// TIA Portal project "MTconnect_V15.1" (V15.1)
// demonstrates certain use cases, when migrating from Rockwell Automation to Siemens

(* hardware
DEVICE "S7-1200 station_1"  S7-1200 Station
   slot 0: "Rack_0"  S7-1200 Rack  Rack  V1.0
   slot 1: "PLC_1"  CPU 1215C AC/DC/Rly  6ES7 215-1BG40-0XB0  V4.1
*)

// ===== PLC "PLC_1"  CPU 1215C AC/DC/Rly =====
// protected blocks, not shown: "MTCONNECT", "TimeStamp"

VAR_GLOBAL   // PLC tag table "Default tag table"
   "Tag_1" AT %M5.5 : Bool;
   "RecDone" AT %M5.0 : Bool;
   "RecBusy" AT %M5.1 : Bool;
   "RecError" AT %M5.2 : Bool;
   "RecStatus" AT %MW6 : Word;
   "RecLength" AT %MW8 : Word;
   "RecTriggerSP" AT %M5.7 : Bool;
   "Clock_Byte" AT %MB0 : Byte;
   "Clock_10Hz" AT %M0.0 : Bool;
   "Clock_5Hz" AT %M0.1 : Bool;
   "Clock_2.5Hz" AT %M0.2 : Bool;
   "Clock_2Hz" AT %M0.3 : Bool;
   "Clock_1.25Hz" AT %M0.4 : Bool;
   "Clock_1Hz" AT %M0.5 : Bool;
   "Clock_0.625Hz" AT %M0.6 : Bool;
   "Clock_0.5Hz" AT %M0.7 : Bool;
   "System_Byte" AT %MB1 : Byte;
   "FirstScan" AT %M1.0 : Bool;
   "DiagStatusUpdate" AT %M1.1 : Bool;
   "AlwaysTRUE" AT %M1.2 : Bool;
   "AlwaysFALSE" AT %M1.3 : Bool;
   "Tag_2" AT %M5.6 : Bool;
   "Tag_3" AT %MD8 : UDInt;
   "Tag_4" AT %M20.0 : Bool;
   "Tag_5" AT %M20.1 : Bool;
   "Tag_6" AT %M20.2 : Bool;
   "Tag_7" AT %MW22 : Word;
   "Tag_8" AT %M20.7 : Bool;
   "Tag_9" AT %M10.7 : Bool;
   "Tag_10" AT %M10.0 : Bool;
   "Tag_11" AT %M10.1 : Bool;
   "Tag_12" AT %M10.2 : Bool;
   "Tag_13" AT %MW12 : Word;
   "SendLength" AT %MW50 : UInt;
   "Tag_15" AT %M50.1 : Bool;
   "Tag_16" AT %M52.1 : Bool;
   "Tag_17" AT %I0.0 : Bool;
   "Tag_18" AT %M15.0 : Bool;
   "SendEvent" AT %M15.1 : Bool;
   "Estop" AT %I0.2 : Bool;
   "Tag_20" AT %M15.2 : Bool;
   "Tag_21" AT %M15.3 : Bool;
   "SendPong" AT %M15.4 : Bool;
   "Tag_22" AT %M15.5 : Bool;
   "Tag_23" AT %M60.0 : Bool;
   "Tag_14" AT %M101.0 : Bool;
   "Tag_24" AT %M21.1 : Bool;
   "Tag_25" AT %MW110 : Word;
   "Tag_26" AT %M109.7 : Bool;
   "InCycle" AT %I0.3 : Bool;
   "Tag_27" AT %I0.4 : Bool;
   "Tag_28" AT %MD16 : DInt;
   "CycleCount" AT %MW20 : Int;
   "Floatnum" AT %MD24 : Real;
END_VAR

VAR_GLOBAL CONSTANT   // PLC tag table "Default tag table"
   "Constant_1" : String := 'This is constant';   // This is Comment
END_VAR

TYPE "DataItemBool"
   STRUCT
      "name" : String[20];
      category : UInt;   // 1) EVENT 2) SAMPLE 3) CONDITION
      value : Bool;
      prevValue : Bool;
      send : Bool;
   END_STRUCT;
END_TYPE

TYPE "DataItemNumeric"
   STRUCT
      "name" : String[20];
      category : UInt;   // 1) EVENT 2) SAMPLE 3) CONDITION
      value : Real;
      prevvalue : Real;
      decimal : Int;
      send : Bool;
   END_STRUCT;
END_TYPE

TYPE "DataItemString"
   STRUCT
      "name" : String[20];
      category : UInt;   // 1) EVENT 2) SAMPLE 3) CONDITION
      value : String[25];
      prevvalue : String[25];
      send : Bool;
   END_STRUCT;
END_TYPE

// folder: MTConnect

DATA_BLOCK "MTCData"   // DB4
{ S7_Optimized_Access := 'TRUE' }
VERSION : 0.1
   VAR
      "Bool" : Array[0..1] of "DataItemBool";
      Numeric : Array[0..1] of "DataItemNumeric";
      "String" : Array[0..1] of "DataItemString";
   END_VAR
BEGIN
   "Bool"[0]."name" := 'estop';
   "Bool"[0].category := 1;   // 1) EVENT 2) SAMPLE 3)CONDITION
   "Bool"[1]."name" := 'btag1';
   "Bool"[0].value := FALSE;
   "Bool"[0].prevValue := FALSE;
   "Bool"[0].send := FALSE;
   "Bool"[1].category := 0;
   "Bool"[1].value := FALSE;
   "Bool"[1].prevValue := FALSE;
   "Bool"[1].send := FALSE;
   Numeric[0]."name" := 'cycles';
   Numeric[0].category := 0;
   Numeric[0].value := 0.0;
   Numeric[0].prevvalue := 0.0;
   Numeric[0].send := FALSE;
   Numeric[1]."name" := 'ftag1';
   Numeric[1].category := 0;
   Numeric[1].value := 0.0;
   Numeric[1].prevvalue := 0.0;
   Numeric[1].send := FALSE;
END_DATA_BLOCK

// folder: (top level)

ORGANIZATION_BLOCK "Main"   // OB1, LAD, ProgramCycle
TITLE = "Main Program Sweep (Cycle)"
{ S7_Optimized_Access := 'TRUE' }
VERSION : 0.1
   VAR_INPUT
      Initial_Call : Bool;   // Initial call of this OB
      Remanence : Bool;   // =True, if remanent data are available
   END_VAR
   VAR_TEMP
      StringTemp1 : String;
      StringTemp2 : String;
   END_VAR
   VAR CONSTANT
      "TRUE/FALSE" : Bool := 1;
   END_VAR
BEGIN

REGION Network 2
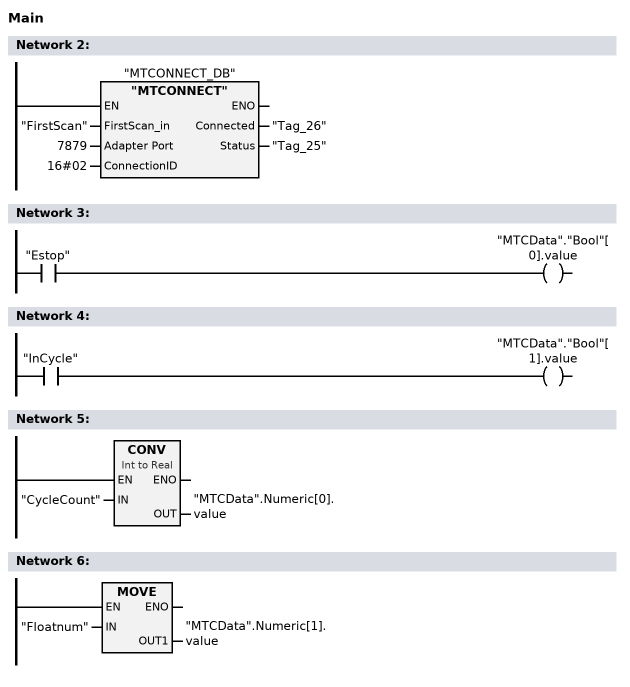
   RUNG wire#powerrail
      "MTCONNECT_DB"(FirstScan_in := "FirstScan", "Adapter Port" := 7879, ConnectionID := 16#02, Connected => "Tag_26", Status => "Tag_25")
   END_RUNG
   // the same network as SCL:
   "MTCONNECT_DB"(FirstScan_in := "FirstScan",   // "MTCONNECT"
                  "Adapter Port" := 7879,
                  ConnectionID := 16#02,
                  Connected => "Tag_26",
                  Status => "Tag_25");
END_REGION

REGION Network 3
   RUNG wire#powerrail
      Contact( "Estop" )
      Coil( "MTCData"."Bool"[0].value )
   END_RUNG
   // the same network as SCL:
   "MTCData"."Bool"[0].value := "Estop";
END_REGION

REGION Network 4
   RUNG wire#powerrail
      Contact( "InCycle" )
      Coil( "MTCData"."Bool"[1].value )
   END_RUNG
   // the same network as SCL:
   "MTCData"."Bool"[1].value := "InCycle";
END_REGION

REGION Network 5
   RUNG wire#powerrail
      { S7_Templates := "[SrcType := Int, DestType := Real]" } Convert(in := "CycleCount", out => "MTCData".Numeric[0].value)
   END_RUNG
   // the same network as SCL:
   "MTCData".Numeric[0].value := INT_TO_REAL("CycleCount");
END_REGION

REGION Network 6
   RUNG wire#powerrail
      Move(in := "Floatnum", out1 => "MTCData".Numeric[1].value)
   END_RUNG
   // the same network as SCL:
   "MTCData".Numeric[1].value := "Floatnum";
END_REGION
END_ORGANIZATION_BLOCK

ORGANIZATION_BLOCK "Data Collection"   // OB30, LAD, CyclicInterrupt
{ S7_Optimized_Access := 'TRUE' }
VERSION : 0.1
   VAR_INPUT
      Initial_Call : Bool;   // Initial call of this OB
      Event_Count : Int;   // Events discarded
   END_VAR
   VAR CONSTANT
      PI : Real := 3.14159;
   END_VAR
BEGIN

REGION Network 2
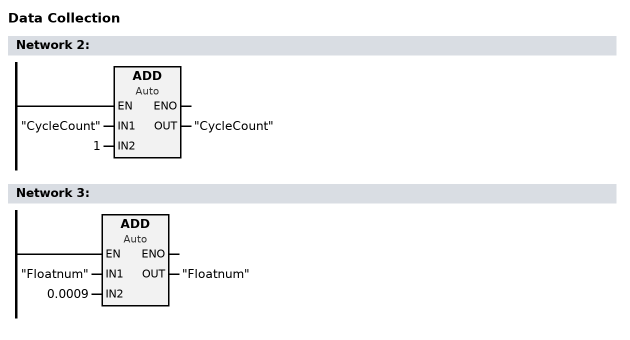
   RUNG wire#powerrail
      Add(in1 := "CycleCount", in2 := 1, out => "CycleCount")
   END_RUNG
   // the same network as SCL:
   "CycleCount" := "CycleCount" + 1;
END_REGION

REGION Network 3
   RUNG wire#powerrail
      Add(in1 := "Floatnum", in2 := 0.0009, out => "Floatnum")
   END_RUNG
   // the same network as SCL:
   "Floatnum" := "Floatnum" + 0.0009;
END_REGION
END_ORGANIZATION_BLOCK

// folder: MTConnect

FUNCTION "SizeOf" : Int   // FC4, SCL
{ S7_Optimized_Access := 'TRUE' }
VERSION : 0.1
   VAR_INPUT
      Arrayin : Variant;
   END_VAR
   VAR_TEMP
      erro : Int;
   END_VAR
BEGIN
   #SizeOf := CountOfElements(#Arrayin);
END_FUNCTION

// ===== library types =====

// folder: GET_PUT_R Datatypes

TYPE "RockwellTag"
VERSION : 0.1
   STRUCT
      ID : Int;   // [INT] TagId inside the remote PLC
      "Name" : String[24];   // [STRING24] TagName inside the remote PLC
      DataType : Int;   // [ENUM] data type of tag
      Count : Int := 1;   // [INT] number of elements to be retrieved
   END_STRUCT;
END_TYPE

TYPE "RockwellTag"
VERSION : 0.1
   STRUCT
      ID : Int;   // [INT] TagId inside the remote PLC
      "Name" : String[24];   // [STRING24] TagName inside the remote PLC
      DataType : Int;   // [ENUM] data type of tag
      Count : Int := 1;   // [INT] number of elements to be retrieved
   END_STRUCT;
END_TYPE

TYPE "RockwellConfig"
VERSION : 0.1
   STRUCT
      connID : Conn_Ouc := 0;   // [1..4096] connection identifier
      currentSessionID : UDInt;   // Session ID used for communications with Rockwell controller / currently used session ID, assigned by the remote PLC
      references : DInt;   // [0..MAX_VAR_R] number of PUT_R/ GET_R instances currently in use / reference count; 0= no connectivity
      instanceLock : DInt;   // instance number currently using send and receive capabilities
   END_STRUCT;
END_TYPE

TYPE "RockwellConfig"
VERSION : 0.1
   STRUCT
      connID : Word;   // [1..4096] connection identifier
      currentSessionID : DInt;   // Session ID used for communications with Rockwell controller / currently used session ID, assigned by the remote PLC
      references : DInt;   // [0..MAX_VAR_R] number of PUT_R/ GET_R instances currently in use / reference count; 0= no connectivity
      instanceLock : DInt;   // instance number currently using send and receive capabilities
   END_STRUCT;
END_TYPE

// folder: (top level)

FUNCTION_BLOCK "PUT_R"   // FB1, SCL
{ S7_Optimized_Access := 'FALSE' }
VERSION : 0.1
   VAR_INPUT
      Enable : Bool;   // [TRUE| FALSE] TRUE signal keeps the block in PowerOff state
      REQ : Bool;   // [TRUE |FALSE] rising edge triggers a read request
      InterfaceId : Byte;   // [1..] InterfaceID of the used interface
      IPv4 : Array[1..4] of Byte;   // [IPv4 address] - shall be in the same subnet as controller is
      Slot : Int;   // [-1..16] -1, when directly connected suc has CompactLogix
   END_VAR
   VAR_OUTPUT
      Status : Word;   // [Enum] status information
      Done : Bool;   // [TRUE | FALSE] TRUE signal is a one shot signal indicating the transmission of the data
      Connecting : Bool;   // [TRUE | FALSE] TRUE signal indicates the establishment of the connection
      Established : Bool;   // [TRUE | FALSE] TRUE indicates an established connection
   END_VAR
   VAR_IN_OUT
      Config : "RockwellConfig";
      Tag : "RockwellTag";   // [RockwelTag] datatype containing the tagname, value and data type
      Value : ANY;
   END_VAR
   VAR
      internalState : Int;   // [Enum] contains the internal state information
      connect : TCON;
      disconnect : TDISCON;
      send : TSEND;
      receive : TRCV;
      connection : TCON_PAR;
      sendBuffer : Struct
         Header : Struct
            Command : Word;   // Encapsulation command
            Length : Int;   // Length, in bytes, of the command specific data portion of the message
            SessionHandle : DInt;   // Session identification
            Status : DInt;   // Status code
            Context : Array[1..8] of Byte;   // Information pertinien only to the sender of an encapsulation command
            Options : DInt;
         END_STRUCT;
         Data : Array[1..508] of Byte;
      END_STRUCT;
      receiveBuffer : Struct
         Header : Struct
            Command : Word;   // Encapsulation command
            Length : Int;   // Length, in bytes, of the command specific data portion of the message
            SessionHandle : DInt;   // Session identification
            Status : DInt;   // Status code
            Context : Array[1..8] of Byte;   // Information pertinien only to the sender of an encapsulation command
            Options : DInt;
         END_STRUCT;
         Data : Array[1..508] of Byte;
      END_STRUCT;
      currentResponse : Word;
      connectionStatus : Struct
         isDisconnected : Bool;
         isDisconnecting : Bool;
         isConnecting : Bool;
         isConnected : Bool;
         hasReceivedData : Bool;
         hasReceivedHeader : Bool;
      END_STRUCT;
      indexTag : Int := 0;
      currentCIPService : Byte;
      previousRequest : Bool;
      EnabledJ : Bool;
      ownInstance : DInt;
      ownSequence : DInt;
      randomGenerator : Struct   // [STRUCT] used to realize a pseudo random number
         m_w : DInt;
         m_z : DInt;
         Val : DInt;
         currentTime : Date_And_Time;
         currentMilliSeconds : Time;
      END_STRUCT;
   END_VAR
   VAR_TEMP
      indexTagName : Int;
      result : Int;
      itemLength : Int;   // contains the Length of the EIP packet
      overallLength : Int;   // contains the Length of the EIP packet
      tagNameLength : Int;   // contains the Length of the Tagname (in WORDS)
      tagValueLength : Int;   // contains the Length of the Tag Value
      unconnectedDataItemLength : Int;   // contains the Length of the unconnected data item
      baseIndexOuterCIPMessage : Int;   // contains the base index to the beginning of the outer CIP message
      baseIndexInnerCIPMessage : Int;   // contains the base index to the beginning of the inner CIP message
      receivedServiceStatus : Int;
      receivedInstance : DInt;
      receivedSequence : DInt;
      receivedType : Word;
      valueIndex : Int;
      bufferIndex : Int;
      tagName : String[24];
      sendValue : Byte;
      DstAny : ANY;
      Destination AT DstAny : Struct
         ID : Byte;
         Typed : Byte;
         Amount : Int;
         Block : Int;
         Offset : Int;
      END_STRUCT;
   END_VAR
   VAR CONSTANT
      EIP_VENDOR_ID : Word := 1251;   // EtherNet/IP vendor ID 'Siemens AG'
      EIP_HEADER_LENGTH : Int := 24;   // EtherNet/IP Encapsulation Header length is 24 bytes
      EIP_PORT : Word := 44818;   // EtherNet/IP standard port is 44818 (0xAF12)
      RESULT_SUCCESS : Word := 16#0000;
      RESULT_IDLE : Word := 16#7000;
      RESULT_JOB_START : Word := 16#7001;
      RESULT_JOB_RUNNING : Word := 16#7002;
      RESULT_JOB_NOT_REQUIRED : Word := 16#80A3;
      RESULT_MORE_AVAIL : Word := 16#80B1;
      RESULT_REUSED_ID : Word := 16#8085;
      EIP_STATUS_OK : DInt := 16#0;   // EIP Status OK
      EIP_STATUS_INVALID_SESSION_ID : DInt := 16#64000000;   // EIP Status "Invalid Session ID"
      EIP_STATUS_TOOMANY_SESSIONS : DInt := 16#01000000;   // EIP Status "more than 1 active session on the same TCP connection"
      EIP_STATUS_OUTOFRESSOURCES : DInt := 16#02000000;   // EIP Status "does not have sufficient resources"
      EIP_STATUS_PROTOCOL_ERROR : DInt := 16#69000000;   // EIP Status "Protocol Version or Options mismatches"
      EIP_CMD_REG_SESSION : Word := 16#0065;   // EtherNet/IP Encapsulation Command "Register Session"
      EIP_CMD_UNREG_SESSION : Word := 16#0066;   // EtherNet/IP Encapsulation Command "Unregister Session"
      EIP_CMD_SEND_RR : Word := 16#006F;   // EtherNet/IP Encapsulation Command "Send RR Data"
      CIP_SRV_TABLEREAD : Byte := 16#4C;   // CIP Service Data Table Read
      CIP_SRV_TABLEWRITE : Byte := 16#4D;   // CIP Service Data Table Write
      CIP_SRV_TABLEREAD_FRAG : Byte := 16#52;   // CIP Service Fragmented Data Table Read
      CIP_SRV_TABLEWRITE_FRAG : Byte := 16#53;   // CIP Service Fragmented Data Table Write
      CIP_SRV_UNCONNECTED_SEND : Byte := 16#52;   // CIP Service Unconnected Send Data
      STATE_IDLE : Int := 1;
      STATE_INIT : Int := 2;
      STATE_CONNECTING : Int := 20;
      STATE_DISCONNECTING : Int := 60;
      STATE_SENDING : Int := 100;
      STATE_REGISTER_SESSION : Int := 22;
      STATE_UNREGISTER_SESSION : Int := 62;
      STATE_REGISTERING : Int := 23;
      STATE_UNREGISTERING : Int := 63;
      STATE_REGISTERED : Int := 24;
      STATE_SEND : Int := 101;
      STATE_RECEIVE_HEADER : Int := 102;
      STATE_RECEIVE_DATA : Int := 103;
      STATE_POWER_OFF : Int := 0;
      DT_BOOLEAN_ATOMIC : Int := 16#C1;
      DT_SINT_ATOMIC : Int := 16#C2;
      DT_INT_ATOMIC : Int := 16#C3;
      DT_DINT_ATOMIC : Int := 16#C4;
      DT_FLOAT_ATOMIC : Int := 16#CA;
      CIP_PATH_SEG_TYPE_CLASS : Byte := 16#20;
      CIP_PATH_SEG_TYPE_INSTANCE : Byte := 16#24;
      CIP_PATH_SEG_TYPE_ANSI : Byte := 16#91;
      CIP_PATH_SEG_TYPE_PORT : Byte := 16#01;
      CIP_ROUTE_SEG_LENGTH : Int := 4;
      CIP_ROUTE_PATH_LENGTH : Int := 1;
      CIP_TABLEREAD_LENGTH : Int := 6;
      CIP_TABLEWRITE_LENGTH : Int := 4;
      CIP_UCSEND_HEADER_LENGTH : Int := 4;
      CIP_UCSEND_SEG_LENGTH : Int := 6;
      EIP_CMD_SEND_RR_SEG_LENGTH : Int := 16;
      CON_TYPE_TCP_V2 : Byte := 16#11;
      CON_TYPE_TCP_V4 : Byte := 11;
      CIP_GENSTS_SUCCESS : Byte := 16#00;
      CIP_GENSTS_PATH_SEG_ERROR : Byte := 16#04;
      CIP_GENSTS_PATH_DEST_UNKNOWN : Byte := 16#05;
      CIP_GENSTS_PARTIAL : Byte := 16#06;
      CIP_GENSTS_NOT_ENOUGH_DATA : Byte := 16#13;
      CIP_GENSTS_PATH_SIZE_MISMATCH : Byte := 16#26;
      CIP_GENSTS_DOESNT_EXIST : Byte := 16#16;
      CIP_GENSTS_GENERIC : Byte := 16#FF;
      CIP_SRVSTS_RANGE_EXCEED : Int := 16#2105;
      CIP_SRVSTS_TYPE_MISMATCH : Int := 16#2107;
   END_VAR
BEGIN
   //=============================================================================
   // Siemens AG
   // (c)Copyright 2016 All Rights Reserved
   //-----------------------------------------------------------------------------
   // Library: PutGet_Rockwell
   // Tested with: 319F-3PN/DP V2.8.6 and ControlLogix/Compactlogix V26
   // Engineering: TIA Portal V13 SP1 Upd 9
   // Restrictions: look into pdf
   // Requirements: 
   // Functionality: Get Put Values from to Rockwell CPU
   //-----------------------------------------------------------------------------
   // Change log table:
   // Version  Date            Expert in charge        Changes applied
   // 01.00.00 12.07.2016      Scheel                  initial version 
   // 01.00.01 20.10.2016      Scheel                  feat: add diagnostics and
   //                                                        indicators
   //                                                  style: remove duplicate
   //                                                         code segments
   //                                                  fix: connect will be
   //                                                       retriggered, when idle
   //                                                  refac: change of IP address
   //                                                         datatype to IP_V4
   //                                                  feat: add recognition of
   //                                                        CIP specific status
   //
   //#########################################################################################
   // Pseudo Random number generator
   //
   //  This Random number function generator is based on multiplication and
   //  addition with overflow invented by George Marsaglia.
   //  The loss of information is intended.
   //  
   //  Wikipedia (https://en.wikipedia.org/wiki/Random_number_generation)
   //#########################################################################################
   //
   //Initialization of the variables using a time value as a seed
   #randomGenerator.currentMilliSeconds := TIME_TCK();

   IF #randomGenerator.m_w = 0 OR #randomGenerator.m_z = 0 THEN
     #randomGenerator.m_w := T_CONV(TIME_TCK());    // using the milliseconds since the PLC has been powered on
     #randomGenerator.m_z := 13696;
   ELSE
     #randomGenerator.m_z := 36969 * DWORD_TO_DINT(DINT_TO_DWORD(#randomGenerator.m_z) AND 16#FFFF)
     + DWORD_TO_DINT(SHR(IN := DINT_TO_DWORD(#randomGenerator.m_z), N := 16));
     #randomGenerator.m_w := 18000 * DWORD_TO_DINT(DINT_TO_DWORD(#randomGenerator.m_w) AND 16#FFFF)
     + DWORD_TO_DINT(SHR(IN := DINT_TO_DWORD(#randomGenerator.m_w), N := 16));
     #randomGenerator.Val := DWORD_TO_DINT(SHL(IN := DINT_TO_DWORD(#randomGenerator.m_z), N := 16)) + #randomGenerator.m_w;  // 32-bit result */    
   END_IF;

   //assume sane state
   #Status := #RESULT_IDLE;
   #Done := FALSE;

   #connect(ID := #connection.id,
            CONNECT := #connection);

   #disconnect(ID := #connection.id);


   IF NOT #Enable AND #EnabledJ THEN
     // Complete Restart detected 
     //
     #internalState := #STATE_UNREGISTER_SESSION;

   ELSIF #Enable AND NOT #EnabledJ THEN
     #internalState := #STATE_INIT;

   ELSE
     // Regular operation
     //   
     CASE #internalState OF
       #STATE_POWER_OFF:
         //Preset the TCP connection information
         //  
         IF #Config.connID = 0 THEN
           #Config.connID := DWORD_TO_WORD(DINT_TO_DWORD((#randomGenerator.Val MOD 2048) + 2048));
         END_IF;
         #connection.id := #Config.connID;

         #connection.connection_type := #CON_TYPE_TCP_V2;      //TCP connection
         #connection.local_device_id := #InterfaceId;
         #connection.active_est := TRUE;                //active connection (Client)

         #connection.local_tsap_id_len := 0;

         #connection.rem_staddr_len := 4;
         #connection.rem_staddr[1] := #IPv4[1];
         #connection.rem_staddr[2] := #IPv4[2];
         #connection.rem_staddr[3] := #IPv4[3];
         #connection.rem_staddr[4] := #IPv4[4];

         #connection.rem_tsap_id_len := 2;
         #connection.rem_tsap_id[1] := WORD_TO_BYTE(SHR(IN := #EIP_PORT, N := 8));
         #connection.rem_tsap_id[2] := WORD_TO_BYTE(#EIP_PORT AND W#16#FF);

         #ownInstance := 0;
         #ownSequence := 0;

         #internalState := #STATE_IDLE;

       #STATE_IDLE:

         // Action
         // 
         #Done := FALSE;

         // Transition 
         //IF NOT #connectionStatus.isConnected THEN
         //  #internalState := #STATE_INIT;          
         IF #connectionStatus.isConnected AND #REQ AND NOT #previousRequest AND #Enable THEN
           #internalState := #STATE_SENDING;
           #Status := #RESULT_JOB_START;
         END_IF;


       #STATE_INIT:
         //Preset the TCP connection information
         //
         IF #Config.connID = 0 THEN
           #Config.connID := DWORD_TO_WORD(DINT_TO_DWORD((#randomGenerator.Val MOD 2048) + 2048));
         END_IF;
         #connection.id := #Config.connID;

         //Inserting Semaphore checking
         //
         //  Only issue a new connect, when there is no one is referencing the connection already
         //  Otherwise just skip that step and use the established connection
         //  

         IF #Config.references = 0 THEN
           #connection.connection_type := #CON_TYPE_TCP_V2;      //TCP connection
           #connection.local_device_id := #InterfaceId;
           #connection.active_est := TRUE;                //active connection (Client)

           #connection.local_tsap_id_len := 0;

           #connection.rem_staddr_len := 4;
           #connection.rem_staddr[1] := #IPv4[1];
           #connection.rem_staddr[2] := #IPv4[2];
           #connection.rem_staddr[3] := #IPv4[3];
           #connection.rem_staddr[4] := #IPv4[4];

           #connection.rem_tsap_id_len := 2;
           #connection.rem_tsap_id[1] := WORD_TO_BYTE(SHR(IN := #EIP_PORT, N := 8));
           #connection.rem_tsap_id[2] := WORD_TO_BYTE(#EIP_PORT AND W#16#FF);


           //No connection established yet
           //  issue a new request
           #connect.REQ := TRUE;
           #internalState := #STATE_CONNECTING;
         ELSE
           #internalState := #STATE_IDLE;
           #connectionStatus.isConnected := TRUE;
         END_IF;
         #Config.references := #Config.references + 1;

         //Remember the currently active instance reference as my own instance identifier
         //  and reset the Sequence counter
         #ownInstance := #Config.references;
         #ownSequence := 0;

       #STATE_CONNECTING:

         IF #connect.STATUS = #RESULT_JOB_START THEN
           #connectionStatus.isConnecting := TRUE;

         ELSIF #connect.STATUS = #RESULT_IDLE THEN
           #connect.REQ := NOT #connect.REQ;

         ELSIF #connect.STATUS = #RESULT_JOB_RUNNING THEN
           #connect.REQ := FALSE;

         ELSIF #connect.STATUS = #RESULT_JOB_NOT_REQUIRED OR
           #connect.STATUS = #RESULT_SUCCESS
         THEN
           #connect.REQ := FALSE;
           #connectionStatus.isConnecting := FALSE;
           #connectionStatus.isConnected := TRUE;
           #connectionStatus.isDisconnected := FALSE;

           #internalState := #STATE_REGISTER_SESSION;

         ELSE
           // Throw error !
           //   Error in connect
           #Status := W#16#8100 OR (#connect.STATUS AND 16#00FF);   //Error in connecting       
           #connect.REQ := FALSE;
           #internalState := #STATE_DISCONNECTING;
         END_IF;

       #STATE_REGISTER_SESSION:

         // SWAP (W#16#AFCD) = W#16#CDAF
         // 
         //  SHL(AFCD, 8) OR SHR(AFCD, 8)

         #sendBuffer.Header.Command := (SHL(IN := #EIP_CMD_REG_SESSION, N := 8) OR SHR(IN := #EIP_CMD_REG_SESSION, N := 8)); //Command is RegisterSession (16#65)
         #sendBuffer.Header.Length := WORD_TO_INT(W#16#0400);          //Length of Data is 4 Bytes
         #sendBuffer.Header.SessionHandle := 0;
         #sendBuffer.Header.Status := 0;
         #sendBuffer.Header.Options := 0;
         //the Context will be a combination out of the own instance identifier
         //and a sequence number
         #sendBuffer.Header.Context[1] := DWORD_TO_BYTE(DINT_TO_DWORD(#ownInstance) AND DW#16#000000FF);
         #sendBuffer.Header.Context[2] := DWORD_TO_BYTE(SHR(IN := DINT_TO_DWORD(#ownInstance), N := 8) AND DW#16#000000FF);
         #sendBuffer.Header.Context[3] := DWORD_TO_BYTE(SHR(IN := DINT_TO_DWORD(#ownInstance), N := 16) AND DW#16#000000FF);
         #sendBuffer.Header.Context[4] := DWORD_TO_BYTE(SHR(IN := DINT_TO_DWORD(#ownInstance), N := 24) AND DW#16#000000FF);
         #sendBuffer.Header.Context[5] := DWORD_TO_BYTE(DINT_TO_DWORD(#ownSequence) AND DW#16#000000FF);
         #sendBuffer.Header.Context[6] := DWORD_TO_BYTE(SHR(IN := DINT_TO_DWORD(#ownSequence), N := 8) AND DW#16#000000FF);
         #sendBuffer.Header.Context[7] := DWORD_TO_BYTE(SHR(IN := DINT_TO_DWORD(#ownSequence), N := 16) AND DW#16#000000FF);
         #sendBuffer.Header.Context[8] := DWORD_TO_BYTE(SHR(IN := DINT_TO_DWORD(#ownSequence), N := 24) AND DW#16#000000FF);
         #sendBuffer.Data[1] := 16#01;                                 //Protocol Version V1.0

         //Checking the MuteEx
         IF #Config.instanceLock = 0 OR
           #Config.instanceLock = #ownInstance
         THEN
           //allowed to utilize, since instanceLock is either 0 or ownInstance
           #send(ID := #connection.id,
                 DATA := #sendBuffer);

           //Locking the MutEx
           #Config.instanceLock := #ownInstance;
           #send.LEN := #EIP_HEADER_LENGTH + 4;
           #send.REQ := TRUE;

           #internalState := #STATE_REGISTERING;
         ELSE
           ;
         END_IF;

       #STATE_REGISTERING:
         // Action
         // 

         //allowed to utilize, since instanceLock is either 0 or ownInstance
         #send(ID := #connection.id,
               DATA := #sendBuffer);

         // Transition
         // 
         IF #send.STATUS = #RESULT_JOB_START THEN
           ;
         ELSIF #send.STATUS = #RESULT_JOB_RUNNING THEN
           #send.REQ := FALSE;

         ELSIF #send.STATUS = #RESULT_IDLE THEN
           #send.REQ := NOT #send.REQ;

         ELSIF #send.STATUS = #RESULT_SUCCESS THEN
           #send.REQ := FALSE;
           #internalState := #STATE_RECEIVE_HEADER;
         ELSE
           // Throw error !
           //   in Registering
           #Status := W#16#8200 OR (#send.STATUS AND 16#00FF);   //Error in sending
           #send.REQ := FALSE;
           #internalState := #STATE_DISCONNECTING;
         END_IF;

       #STATE_SENDING:
         #sendBuffer.Header.Command := (SHL(IN := #EIP_CMD_SEND_RR, N := 8) OR SHR(IN := #EIP_CMD_SEND_RR, N := 8));       //Command is SendRRData (16#6F)
         //
         // overall Message length depends on the packet content and is therefore assigned later
         //
         // SWAP (DW#16#0102ABCD) = CDAB0201
         // 
         //   = SHL(<value>,24) OR (SHL(<value>, 8) AND DW#16#00FF0000) OR (SHR(<value>, 8) AND DW#16#0000FF00) OR SHR(<value>,24)

         //#sendBuffer.Header.SessionHandle := DWORD_TO_DINT(SWAP(DINT_TO_DWORD(#Config.currentSessionID)));
         #sendBuffer.Header.SessionHandle := DWORD_TO_DINT(SHL(IN := DINT_TO_DWORD(#Config.currentSessionID), N := 24) OR
                                                           (SHL(IN := DINT_TO_DWORD(#Config.currentSessionID), N := 8) AND DW#16#00FF0000) OR
                                                           (SHR(IN := DINT_TO_DWORD(#Config.currentSessionID), N := 8) AND DW#16#0000FF00) OR
                                                           SHR(IN := DINT_TO_DWORD(#Config.currentSessionID), N := 24));

         ;
         #sendBuffer.Header.Status := 0;
         #sendBuffer.Header.Options := 0;
         //the Context will be a combination out of the own instance identifier
         //and a sequence number
         #sendBuffer.Header.Context[1] := DWORD_TO_BYTE(DINT_TO_DWORD(#ownInstance) AND DW#16#000000FF);
         #sendBuffer.Header.Context[2] := DWORD_TO_BYTE(SHR(IN := DINT_TO_DWORD(#ownInstance), N := 8) AND DW#16#000000FF);
         #sendBuffer.Header.Context[3] := DWORD_TO_BYTE(SHR(IN := DINT_TO_DWORD(#ownInstance), N := 16) AND DW#16#000000FF);
         #sendBuffer.Header.Context[4] := DWORD_TO_BYTE(SHR(IN := DINT_TO_DWORD(#ownInstance), N := 24) AND DW#16#000000FF);
         #sendBuffer.Header.Context[5] := DWORD_TO_BYTE(DINT_TO_DWORD(#ownSequence) AND DW#16#000000FF);
         #sendBuffer.Header.Context[6] := DWORD_TO_BYTE(SHR(IN := DINT_TO_DWORD(#ownSequence), N := 8) AND DW#16#000000FF);
         #sendBuffer.Header.Context[7] := DWORD_TO_BYTE(SHR(IN := DINT_TO_DWORD(#ownSequence), N := 16) AND DW#16#000000FF);
         #sendBuffer.Header.Context[8] := DWORD_TO_BYTE(SHR(IN := DINT_TO_DWORD(#ownSequence), N := 24) AND DW#16#000000FF);
         //CIP specific data
         #sendBuffer.Data[1] := 16#0;                                 //CIP Interface handle
         #sendBuffer.Data[2] := 16#0;
         #sendBuffer.Data[3] := 16#0;
         #sendBuffer.Data[4] := 16#0;

         #sendBuffer.Data[5] := 16#0;                                  //Timeout
         #sendBuffer.Data[6] := 16#0;

         #sendBuffer.Data[7] := 16#2;                                  //Items
         #sendBuffer.Data[8] := 16#0;

         #sendBuffer.Data[9] := 16#0;                                  //Null address item
         #sendBuffer.Data[10] := 16#0;
         #sendBuffer.Data[11] := 16#0;                                  //Null address item Length = 0
         #sendBuffer.Data[12] := 16#0;

         #sendBuffer.Data[13] := 16#B2;                                  //Unconnected data item
         #sendBuffer.Data[14] := 16#0;
         //Item Length needs to be added, but since that depends on the content,
         //it will will be assigned later. It occupies 2 Bytes, thus the outer CIP Message 
         //starts at offset 17 into the Data (1 based counting)
         //
         #baseIndexOuterCIPMessage := 17;

         //CIP Message
         //  here a decision needs to be made
         //  In case Slot is -1 a direct connection is assumed, such as for a CompactLogix, this means no
         //  further route segments are necessary
         //  In case Slot is anywhere between 0 and 16 a route segment is required, since the CPU is not
         //  identical to the ethernet interface, as in a ControlLogix L5, L6, L7 series system

         //Length of the following Path segment depends only on the length of the Tagname measured in WORDS
         // plus 1 WORD for the segment encoding information
         // 
         #tagName := #Tag."Name";
         #tagNameLength := ((LEN(#tagName) + 1) / 2) * 2;

         //
         //  Prelude
         //
         //In case the slot information is negative (-1) there is no additional path segment
         //Any other slot value requires routing information, which need to be added
         //  this means the preparation of offsets and header needs to be done, before
         //  the common part of copying the value to the packet can take place
         IF #Slot = -1 THEN
           //directly connected (onboard) Ethernet interface
           //
           #baseIndexInnerCIPMessage := #baseIndexOuterCIPMessage;

         ELSE
           //not directly connected (through external) Ethernet interface
           //
           //  preparing offsets for length calculation as well as header
           //  There is a 10 byte segment before the tag value segment
           #baseIndexInnerCIPMessage := #baseIndexOuterCIPMessage + 10;

           #sendBuffer.Data[#baseIndexOuterCIPMessage] := #CIP_SRV_UNCONNECTED_SEND;                //CIP service = UNCONNECTED_SEND_DATA = 16#52
           #sendBuffer.Data[#baseIndexOuterCIPMessage + 1] := 2;                                    //Path Size is constant 2 WORDS

           #sendBuffer.Data[#baseIndexOuterCIPMessage + 2] := #CIP_PATH_SEG_TYPE_CLASS;             //Path Type = Class Segment
           #sendBuffer.Data[#baseIndexOuterCIPMessage + 3] := 16#06;                                //Class = ConnectionManager (16#06)

           #sendBuffer.Data[#baseIndexOuterCIPMessage + 4] := #CIP_PATH_SEG_TYPE_INSTANCE;          //Path Type = Instance Segment
           #sendBuffer.Data[#baseIndexOuterCIPMessage + 5] := 16#01;                                //Instance =Instance 1 (16#01)

           //Encapsulated CIP Message
           //
           #sendBuffer.Data[#baseIndexOuterCIPMessage + 6] := 16#07;                                //Priority combined with TimeTick (= 16#07)
           #sendBuffer.Data[#baseIndexOuterCIPMessage + 7] := INT_TO_BYTE(233);                     //???

         END_IF;

         //
         // tag value segment
         // 

         #sendBuffer.Data[#baseIndexInnerCIPMessage] := #CIP_SRV_TABLEWRITE;                        //CIP service = DATA_TABLE_READ = 16#4D

         #sendBuffer.Data[#baseIndexInnerCIPMessage + 1] := DINT_TO_BYTE(#tagNameLength / 2 + 1);  //Path Size
         #sendBuffer.Data[#baseIndexInnerCIPMessage + 2] := #CIP_PATH_SEG_TYPE_ANSI;                //Path Type = ANSI Extended Symbol Segment

         //Copy In
         //
         #tagName := #Tag."Name";
         #sendBuffer.Data[#baseIndexInnerCIPMessage + 3] := INT_TO_BYTE(LEN(#tagName));   //TagName Length (bytes)
         FOR #indexTagName := 1 TO BYTE_TO_INT(#sendBuffer.Data[#baseIndexInnerCIPMessage + 3]) DO
           #sendBuffer.Data[#baseIndexInnerCIPMessage + 3 + #indexTagName] := CHAR_TO_BYTE(S_CONV(MID(IN := #tagName, L := 1, P := #indexTagName)));
         END_FOR;
         //in case the tag name has an odd (uneven) length the path segment content needs to be padded to be WORD aligned
         //
         #indexTagName := #indexTagName - 1;
         IF #indexTagName MOD 2 <> 0 THEN
           #indexTagName := #indexTagName + 1;
           #sendBuffer.Data[#baseIndexInnerCIPMessage + 3 + #indexTagName] := 0;
         END_IF;

         //Command Specific information
         //
         #sendBuffer.Data[#baseIndexInnerCIPMessage + 4 + #indexTagName] := INT_TO_BYTE(#Tag.DataType);
         #sendBuffer.Data[#baseIndexInnerCIPMessage + 5 + #indexTagName] := 0;
         #sendBuffer.Data[#baseIndexInnerCIPMessage + 6 + #indexTagName] := INT_TO_BYTE(#Tag.Count);                 //number of values to follow
         #sendBuffer.Data[#baseIndexInnerCIPMessage + 7 + #indexTagName] := WORD_TO_BYTE(SHR(IN := INT_TO_WORD(#Tag.Count), N := 8) AND W#16#00FF);

         #bufferIndex := #baseIndexInnerCIPMessage + 8 + #indexTagName;

         #DstAny := #sendBuffer.Data[#bufferIndex];
         #Destination.Amount := #Tag.Count;

         //Copy the value in, type dependant
         CASE #Tag.DataType OF
           #DT_BOOLEAN_ATOMIC:
             //Transferring the Value
             //
             // Adjust the type
             #Destination.Typed := B#16#02;


             #result := BLKMOV(SRCBLK := #Value,
                               DSTBLK => #DstAny);

             #tagValueLength := 4 + #Tag.Count * 1;
           #DT_SINT_ATOMIC:
             //Transferring the Value
             //
             // Adjust the type
             #Destination.Typed := B#16#02;

             #result := BLKMOV(SRCBLK := #Value,
                               DSTBLK => #DstAny);
             #tagValueLength := 4 + #Tag.Count * 1;
           #DT_INT_ATOMIC:
             //Transferring the Value
             //
             // Adjust the type
             #Destination.Typed := B#16#05;

             #result := BLKMOV(SRCBLK := #Value,
                               DSTBLK => #DstAny);

             // Swapping the bytes for each value
             // 
             #valueIndex := 0;

             WHILE #valueIndex <= #Tag.Count DO
               #sendValue                                           := #sendBuffer.Data[#bufferIndex + 1 + 2 * #valueIndex];
               #sendBuffer.Data[#bufferIndex + 1 + 2 * #valueIndex] := #sendBuffer.Data[#bufferIndex     + 2 * #valueIndex];
               #sendBuffer.Data[#bufferIndex     + 2 * #valueIndex] := #sendValue;
               #valueIndex := #valueIndex + 1;
             END_WHILE;

             #tagValueLength := 4 + #Tag.Count * 2;
           #DT_DINT_ATOMIC:
             //Transferring the Value
             //
             // Adjust the type
             #Destination.Typed := B#16#07;

             #result := BLKMOV(SRCBLK := #Value,
                               DSTBLK => #DstAny);

             #valueIndex := 0;
             WHILE #valueIndex <= #Tag.Count DO

               // swap the received value
               #sendValue                                           := #sendBuffer.Data[#bufferIndex + 3 + 2 * #valueIndex];
               #sendBuffer.Data[#bufferIndex + 3 + 2 * #valueIndex] := #sendBuffer.Data[#bufferIndex     + 2 * #valueIndex];
               #sendBuffer.Data[#bufferIndex     + 2 * #valueIndex] := #sendValue;

               #sendValue                                           := #sendBuffer.Data[#bufferIndex + 2 + 2 * #valueIndex];
               #sendBuffer.Data[#bufferIndex + 2 + 2 * #valueIndex] := #sendBuffer.Data[#bufferIndex + 1 + 2 * #valueIndex];
               #sendBuffer.Data[#bufferIndex + 1 + 2 * #valueIndex] := #sendValue;

               #valueIndex := #valueIndex + 1;
             END_WHILE;

             #tagValueLength := 4 + #Tag.Count * 4;
           #DT_FLOAT_ATOMIC:
             //Transferring the Value
             //
             // Adjust the type
             #Destination.Typed := B#16#08;

             #result := BLKMOV(SRCBLK := #Value,
                               DSTBLK => #DstAny);

             #valueIndex := 0;
             WHILE #valueIndex <= #Tag.Count DO

               // swap the received value
               #sendValue                                           := #sendBuffer.Data[#bufferIndex + 3 + 2 * #valueIndex];
               #sendBuffer.Data[#bufferIndex + 3 + 2 * #valueIndex] := #sendBuffer.Data[#bufferIndex     + 2 * #valueIndex];
               #sendBuffer.Data[#bufferIndex     + 2 * #valueIndex] := #sendValue;

               #sendValue                                           := #sendBuffer.Data[#bufferIndex + 2 + 2 * #valueIndex];
               #sendBuffer.Data[#bufferIndex + 2 + 2 * #valueIndex] := #sendBuffer.Data[#bufferIndex + 1 + 2 * #valueIndex];
               #sendBuffer.Data[#bufferIndex + 1 + 2 * #valueIndex] := #sendValue;

               #valueIndex := #valueIndex + 1;
             END_WHILE;

             #tagValueLength := 4 + #Tag.Count * 4;
         ELSE

           //Throw error
           //  - unknown/ unsupported data type specified
           //  
           // throw warning
           #Status := 16#71A3; //Unknown data type
           #tagValueLength := 0;
         END_CASE;

         #itemLength := #tagNameLength + #tagValueLength + #CIP_TABLEWRITE_LENGTH;

         //
         // Closure
         //

         IF #Slot = -1 THEN
           #unconnectedDataItemLength := #itemLength;
         ELSE
           #sendBuffer.Data[#baseIndexOuterCIPMessage + 8] := WORD_TO_BYTE(DINT_TO_WORD(#itemLength));                  //Unconnected data item Length
           #sendBuffer.Data[#baseIndexOuterCIPMessage + 9] := WORD_TO_BYTE(SHL(IN := DINT_TO_WORD(#itemLength), N := 8));  //Unconnected data item Length

           //Routing Information
           #sendBuffer.Data[#baseIndexInnerCIPMessage + #itemLength] := INT_TO_BYTE(#CIP_ROUTE_PATH_LENGTH);
           #sendBuffer.Data[#baseIndexInnerCIPMessage + #itemLength + 1] := 0;

           #sendBuffer.Data[#baseIndexInnerCIPMessage + #itemLength + 2] := #CIP_PATH_SEG_TYPE_PORT;
           #sendBuffer.Data[#baseIndexInnerCIPMessage + #itemLength + 3] := INT_TO_BYTE(#Slot);



           #unconnectedDataItemLength :=   #itemLength
                                         + #CIP_ROUTE_SEG_LENGTH
                                         + #CIP_UCSEND_HEADER_LENGTH
                                         + #CIP_UCSEND_SEG_LENGTH;
         END_IF;

         //Length of the unconnected data item depends on the content of the package
         //
         #sendBuffer.Data[15] := WORD_TO_BYTE(DINT_TO_WORD(#unconnectedDataItemLength));        //Unconnected data item Length
         #sendBuffer.Data[16] := WORD_TO_BYTE(SHL(IN := DINT_TO_WORD(#unconnectedDataItemLength), N := 8));  //Unconnected data item Length


         #sendBuffer.Header.Length := WORD_TO_INT(SHL(IN := INT_TO_WORD(#unconnectedDataItemLength + #EIP_CMD_SEND_RR_SEG_LENGTH), N := 8) OR
                                                  SHR(IN := INT_TO_WORD(#unconnectedDataItemLength + #EIP_CMD_SEND_RR_SEG_LENGTH), N := 8));    //Length of Data

         //Checking the MuteEx
         IF #Config.instanceLock = 0 OR
           #Config.instanceLock = #ownInstance
         THEN
           #Config.instanceLock := #ownInstance;
           #send.LEN := DINT_TO_INT(#EIP_HEADER_LENGTH + #unconnectedDataItemLength + #EIP_CMD_SEND_RR_SEG_LENGTH);
           #send.REQ := TRUE;

           #ownSequence := #ownSequence + 1;
           //allowed to utilize, since instanceLock is either 0 or ownInstance
           #send(ID := #connection.id,
                 DATA := #sendBuffer);

           #internalState := #STATE_SEND;
         ELSE
           ;
         END_IF;
         #Status := #RESULT_JOB_RUNNING;

       #STATE_SEND:
         // Action
         // 

         // assume job is still running
         #Status := #RESULT_JOB_RUNNING;

         #send(ID := #connection.id,
               DATA := #sendBuffer);

         // Transition
         //
         IF #send.STATUS = #RESULT_JOB_START THEN
           ;
         ELSIF #send.STATUS = #RESULT_IDLE THEN
           #send.REQ := NOT #send.REQ;

         ELSIF #send.STATUS = #RESULT_JOB_RUNNING THEN
           #send.REQ := FALSE;

         ELSIF #send.STATUS = #RESULT_SUCCESS THEN
           #send.REQ := FALSE;
           #internalState := #STATE_RECEIVE_HEADER;
         ELSE
           // Throw error !
           // 
            #Status := W#16#8200 OR (#send.STATUS AND 16#00FF);
           #send.REQ := FALSE;
           #internalState := #STATE_DISCONNECTING;
         END_IF;

       #STATE_RECEIVE_HEADER:
         // Action
         // Receive Header data
         // 

         // assume job is still running
         #Status := #RESULT_JOB_RUNNING;

         #receive(EN_R := (#ownInstance = #Config.instanceLock),
                  ID := #connection.id,
                  LEN := #EIP_HEADER_LENGTH,
                  DATA := #receiveBuffer.Header);


         // Transition
         // Header received --> STATE_RECEIVE_DATA
         // Invalid Data --> IDLE
         // Error --> INIT
         IF #receive.NDR OR #receive.STATUS = #RESULT_SUCCESS THEN
           IF #receiveBuffer.Header.Length = 0 THEN
             //Unlocking MuteEx
             #Config.instanceLock := 0;
             #internalState := #STATE_IDLE;
           ELSE
             #internalState := #STATE_RECEIVE_DATA;
           END_IF;
         ELSIF #receive.STATUS <> #RESULT_IDLE AND
           #receive.STATUS <> #RESULT_JOB_RUNNING AND
           #receive.STATUS <> #RESULT_JOB_START AND
           #receive.STATUS <> #RESULT_SUCCESS
         THEN
           #Status := W#16#8300 OR (#receive.STATUS AND 16#00FF);
           #internalState := #STATE_IDLE;
         ELSE
           //Nothing to do, just wait here
           ;
         END_IF;

       #STATE_RECEIVE_DATA:
         // Action
         // Receive Data
         // 
         // assume job is still running
         #Status := #RESULT_JOB_RUNNING;

         #receive(EN_R := (#ownInstance = #Config.instanceLock),
                  ID := #connection.id,
                  LEN := WORD_TO_INT((SHL(IN:=INT_TO_WORD(#receiveBuffer.Header.Length),N:= 8) OR
                                      SHR(IN:=INT_TO_WORD(#receiveBuffer.Header.Length),N:= 8))),
                  DATA := #receiveBuffer.Data);

         // Transition
         // Header received --> STATE_RECEIVE_DATA
         // Invalid Data --> IDLE
         // Error --> INIT
         IF #receive.NDR OR #receive.STATUS = #RESULT_SUCCESS THEN
           // Decode Response
           // 
           #currentResponse := (SHL(IN:=#receiveBuffer.Header.Command, N:=8) OR
                                SHR(IN:=#receiveBuffer.Header.Command, N:=8));

           //the Context will be a combination out of the own instance identifier
           //and a sequence number
           #receivedInstance := DWORD_TO_DINT(SHL(IN := BYTE_TO_DWORD(#receiveBuffer.Header.Context[4]), N := 24) OR
                                              SHL(IN := BYTE_TO_DWORD(#receiveBuffer.Header.Context[3]), N := 16) OR
                                              SHL(IN := BYTE_TO_DWORD(#receiveBuffer.Header.Context[2]), N := 8) OR
                                              BYTE_TO_DWORD(#receiveBuffer.Header.Context[1]));

           #receivedSequence := DWORD_TO_DINT(SHL(IN := BYTE_TO_DWORD(#receiveBuffer.Header.Context[8]), N := 24) OR
                                              SHL(IN := BYTE_TO_DWORD(#receiveBuffer.Header.Context[7]), N := 16) OR
                                              SHL(IN := BYTE_TO_DWORD(#receiveBuffer.Header.Context[6]), N := 8) OR
                                              BYTE_TO_DWORD(#receiveBuffer.Header.Context[5]));

           IF #currentResponse = #EIP_CMD_REG_SESSION THEN
             //Response to RegisterSession received
             // retrieve the SessionID (SessionHandle)
             IF #receiveBuffer.Header.Status = #EIP_STATUS_OK THEN
               #Config.currentSessionID := DWORD_TO_DINT(SHL(IN := DINT_TO_DWORD(#receiveBuffer.Header.SessionHandle), N := 24) OR
                                                         (SHL(IN := DINT_TO_DWORD(#receiveBuffer.Header.SessionHandle), N := 8) AND DW#16#00FF0000) OR
                                                         (SHR(IN := DINT_TO_DWORD(#receiveBuffer.Header.SessionHandle), N := 8) AND DW#16#0000FF00) OR
                                                         SHR(IN := DINT_TO_DWORD(#receiveBuffer.Header.SessionHandle), N := 24));
               #Status := #RESULT_SUCCESS;
             ELSE
               // inform the user about it
               //
               #Status := W#16#7100 OR DWORD_TO_WORD((SHR(IN := DINT_TO_DWORD(#receiveBuffer.Header.Status), N := 24)));

               //Cleaning up internal information and
               //gracefully disconnect
               IF #Config.currentSessionID = 0 THEN
                 // a previous session hasn't been established --> only disconnecting
                 #internalState := #STATE_DISCONNECTING;
               ELSE
                 // previous session existed (somehow) --> unregister before disconnecting
                 #internalState := #STATE_UNREGISTER_SESSION;
               END_IF;
             END_IF;

           ELSIF #currentResponse = #EIP_CMD_SEND_RR THEN
             //Response to Send RR Data received
             // determine Status of transmission
             // retrieve TagValue and DataType
             IF #receiveBuffer.Header.Status = #EIP_STATUS_OK THEN
               #itemLength := WORD_TO_INT(SHL(IN := BYTE_TO_WORD(#receiveBuffer.Data[16]), N := 8) OR BYTE_TO_WORD(#receiveBuffer.Data[15]));
               #currentCIPService := #receiveBuffer.Data[17];
               IF #currentCIPService = (#CIP_SRV_TABLEWRITE OR 16#80) AND
                 #receivedInstance = #ownInstance AND
                 #receivedSequence = #ownSequence
               THEN
                 #ownSequence := #ownSequence + 1;

                 IF #receiveBuffer.Data[19] = #CIP_GENSTS_SUCCESS THEN
                   #Status := #RESULT_SUCCESS;
                   #Done := TRUE;

                 ELSIF #receiveBuffer.Data[19] = #CIP_GENSTS_PATH_DEST_UNKNOWN OR
                       #receiveBuffer.Data[19] = #CIP_GENSTS_PATH_SEG_ERROR
                 THEN
                   // throw warning
                   #Status := W#16#7200 OR #receiveBuffer.Data[19];

                 ELSIF #receiveBuffer.Data[19] = #CIP_GENSTS_GENERIC THEN
                   #Status := W#16#7300 OR #receiveBuffer.Data[21];
                 ELSE
                   // throw warning
                   #Status := W#16#72FF;  //Unknown error code
                 END_IF;

               ELSIF #currentCIPService = (#CIP_SRV_TABLEWRITE_FRAG OR 16#80) THEN
                 #Status := W#16#7300 OR #receiveBuffer.Data[19];

               ELSE
                 // throw warning
                 //   unexpected answer from host - ignoring it
                 #Status := W#16#8A00 OR #currentCIPService;
               END_IF;

             ELSE
               // inform the user about it
               //
               #Status := W#16#7100 OR DWORD_TO_WORD((SHR(IN := DINT_TO_DWORD(#receiveBuffer.Header.Status), N := 24)));

               //Cleaning up internal information and
               //gracefully disconnect
               IF #Config.currentSessionID = 0 THEN
                   // a previous session hasn't been established --> only disconnecting
                   #internalState := #STATE_DISCONNECTING;
                 ELSE
                   // previous session existed (somehow) --> unregister before disconnecting
                   #internalState := #STATE_UNREGISTER_SESSION;
                 END_IF;
             END_IF;
           ELSE
             //Unknown/ Unhandled Response received
             //  ignoring it
             #Status := W#16#8B00 OR #currentResponse;
             //#Config.currentSessionID := 0;
             //#internalState := #STATE_DISCONNECTING;
           END_IF;

           #receiveBuffer.Header.Length := 0;

           //Unlocking MuteEx
           #Config.instanceLock := 0;

           #internalState := #STATE_IDLE;

         ELSIF #receive.STATUS <> #RESULT_IDLE AND
           #receive.STATUS <> #RESULT_JOB_RUNNING AND
           #receive.STATUS <> #RESULT_JOB_START AND
           #receive.STATUS <> #RESULT_SUCCESS
         THEN
           #Status := W#16#8300 OR (#receive.STATUS AND 16#00FF);
           #internalState := #STATE_IDLE;
         ELSE
           ;
         END_IF;

       #STATE_UNREGISTER_SESSION:
         IF #Config.references = 1 THEN

           #sendBuffer.Header.Command := SHL(IN := #EIP_CMD_UNREG_SESSION, N := 8) OR
           SHR(IN := #EIP_CMD_UNREG_SESSION, N := 8);   //Command is RegisterSession (16#66)
           #sendBuffer.Header.Length := WORD_TO_INT(SHL(IN := INT_TO_WORD(#send.LEN - #EIP_HEADER_LENGTH), N := 8) OR
                                                    SHR(IN := INT_TO_WORD(#send.LEN - #EIP_HEADER_LENGTH), N := 8));    //Length of Data is 4 Bytes

           // SWAP (DW#16#0102ABCD) = CDAB0201
           // 
           //   = SHL(<value>,24) OR (SHL(<value>, 8) AND DW#16#00FF0000) OR (SHR(<value>, 8) AND DW#16#0000FF00) OR SHR(<value>,24)

           //#sendBuffer.Header.SessionHandle := DWORD_TO_DINT(SWAP(DINT_TO_DWORD(#Config.currentSessionID)));
           #sendBuffer.Header.SessionHandle := DWORD_TO_DINT(SHL(IN := DINT_TO_DWORD(#Config.currentSessionID), N := 24) OR
                                                             (SHL(IN := DINT_TO_DWORD(#Config.currentSessionID), N := 8) AND DW#16#00FF0000) OR
                                                             (SHR(IN := DINT_TO_DWORD(#Config.currentSessionID), N := 8) AND DW#16#0000FF00) OR
                                                             SHR(IN := DINT_TO_DWORD(#Config.currentSessionID), N := 24));
           #sendBuffer.Header.Status := 0;
           #sendBuffer.Header.Options := 0;
           //the Context will be a combination out of the own instance identifier
           //and a sequence number
           #sendBuffer.Header.Context[1] := DWORD_TO_BYTE(DINT_TO_DWORD(#ownInstance) AND DW#16#000000FF);
           #sendBuffer.Header.Context[2] := DWORD_TO_BYTE(SHR(IN := DINT_TO_DWORD(#ownInstance), N := 8) AND DW#16#000000FF);
           #sendBuffer.Header.Context[3] := DWORD_TO_BYTE(SHR(IN := DINT_TO_DWORD(#ownInstance), N := 16) AND DW#16#000000FF);
           #sendBuffer.Header.Context[4] := DWORD_TO_BYTE(SHR(IN := DINT_TO_DWORD(#ownInstance), N := 24) AND DW#16#000000FF);
           #sendBuffer.Header.Context[5] := DWORD_TO_BYTE(DINT_TO_DWORD(#ownSequence) AND DW#16#000000FF);
           #sendBuffer.Header.Context[6] := DWORD_TO_BYTE(SHR(IN := DINT_TO_DWORD(#ownSequence), N := 8) AND DW#16#000000FF);
           #sendBuffer.Header.Context[7] := DWORD_TO_BYTE(SHR(IN := DINT_TO_DWORD(#ownSequence), N := 16) AND DW#16#000000FF);
           #sendBuffer.Header.Context[8] := DWORD_TO_BYTE(SHR(IN := DINT_TO_DWORD(#ownSequence), N := 24) AND DW#16#000000FF);
           #sendBuffer.Data[1] := 16#00;

           //Checking the MuteEx
           IF #Config.instanceLock = 0 OR
             #Config.instanceLock = #ownInstance
           THEN
             //Locking the MutEx
             #Config.instanceLock := #ownInstance;
             #send.LEN := #EIP_HEADER_LENGTH;
             #send.REQ := TRUE;
             // Action
             // 

             #send(ID := #connection.id,
                   DATA := #sendBuffer);

             // Transition
             //
             #internalState := #STATE_UNREGISTERING;
             #Config.references := #Config.references - 1;
           ELSE
             IF #Config.instanceLock = #ownInstance THEN
               #Config.instanceLock := 0;
             END_IF;
           END_IF;
         ELSE
           IF #Config.references > 1 THEN
             #Config.references := #Config.references - 1;
           END_IF;
           #internalState := #STATE_POWER_OFF;
         END_IF;

       #STATE_UNREGISTERING:
         // Action
         // 

         #send(ID := #connection.id,
               DATA := #sendBuffer);

         // Transition
         //
         IF #send.STATUS = #RESULT_JOB_START THEN
           ;
         ELSIF #send.STATUS = #RESULT_JOB_RUNNING THEN
           #send.REQ := FALSE;

         ELSIF #send.STATUS = #RESULT_IDLE THEN
           #send.REQ := NOT #send.REQ;

         ELSIF #send.STATUS = #RESULT_SUCCESS THEN
           #send.REQ := FALSE;
           #internalState := #STATE_DISCONNECTING;
           //Unlocking MuteEx
           #Config.instanceLock := 0;

         ELSE
           // Throw error !
           //   Error from Sending
           #Status := W#16#8200 OR (#send.STATUS AND 16#00FF);
           #send.REQ := FALSE;
           #internalState := #STATE_DISCONNECTING;
         END_IF;

       #STATE_DISCONNECTING:

         IF #disconnect.STATUS = #RESULT_JOB_START THEN
           #connectionStatus.isConnected := FALSE;
           #connectionStatus.isDisconnecting := TRUE;

         ELSIF #disconnect.STATUS = #RESULT_IDLE THEN
           #connectionStatus.isDisconnecting := TRUE;
           #disconnect.REQ := NOT #disconnect.REQ;

         ELSIF #disconnect.STATUS = #RESULT_JOB_RUNNING THEN
           #disconnect.REQ := FALSE;

         ELSIF #disconnect.STATUS = #RESULT_JOB_NOT_REQUIRED OR
           #disconnect.STATUS = #RESULT_SUCCESS
         THEN
           #disconnect.REQ := FALSE;
           #connectionStatus.isConnected := FALSE;
           #connectionStatus.isDisconnecting := FALSE;
           #connectionStatus.isDisconnected := TRUE;
           #connectionStatus.hasReceivedData := FALSE;
           #connectionStatus.hasReceivedHeader := FALSE;
           //#Config.currentSessionID := 0;
           #ownInstance := 0;
           #ownSequence := 0;
           #Config.connID := 0;

           #internalState := #STATE_IDLE;
         ELSE
           // Throw error !
           //   Error from disconnecting
           #Status := W#16#8400 OR (#disconnect.STATUS AND 16#00FF);
           #disconnect.REQ := FALSE;
           #connectionStatus.isConnected := FALSE;
           #connectionStatus.isDisconnecting := FALSE;
           #connectionStatus.isDisconnected := TRUE;
           #connectionStatus.hasReceivedData := FALSE;
           #connectionStatus.hasReceivedHeader := FALSE;

           //#Config.currentSessionID := 0;
           #ownInstance := 0;
           #ownSequence := 0;

           #internalState := #STATE_IDLE;

         END_IF;
       ELSE
         // Throw error !
         //   unknown internal state        
         #Status := W#16#8C00 OR (INT_TO_WORD(#internalState) AND W#16#00FF);
     END_CASE;
   END_IF;

   #previousRequest := #REQ;
   #EnabledJ := #Enable;
END_FUNCTION_BLOCK

FUNCTION_BLOCK "GET_R"   // FB2, SCL
{ S7_Optimized_Access := 'FALSE' }
VERSION : 0.1
   VAR_INPUT
      Enable : Bool;   // [TRUE| FALSE] TRUE signal keeps the block in PowerOff state
      REQ : Bool;   // [TRUE |FALSE] rising edge triggers a read request
      InterfaceId : Byte;   // [1..] InterfaceID of the used interface
      IPv4 : Array[1..4] of Byte;   // [IP v4 address] IP address of the remote rack
      Slot : Int;   // [-1..16] Slot the addressed CPU is located; -1 if directly connected
   END_VAR
   VAR_OUTPUT
      Status : Word;   // [Enum] status information
      NewData : Bool;   // [TRUE | FALSE] TRUE signal is a one shot signal indicating the receiption of the requested data
      Connecting : Bool;   // [TRUE | FALSE] TRUE signal indicates the establishment of the connection
      Established : Bool;   // [TRUE | FALSE] TRUE indicates an established connection
   END_VAR
   VAR_IN_OUT
      Config : "RockwellConfig";
      Tag : "RockwellTag";   // [RockwelTag] datatype containing the tagname, value and data type
      Value : ANY;
   END_VAR
   VAR
      internalState : Int;   // [Enum] contains the internal state information
      connect : TCON;
      disconnect : TDISCON;
      send : TSEND;
      receive : TRCV;
      connection : TCON_PAR;
      sendBuffer : Struct
         Header : Struct
            Command : Word;   // Encapsulation command
            Length : Int;   // Length, in bytes, of the command specific data portion of the message
            SessionHandle : DInt;   // Session identification
            Status : DInt;   // Status code
            Context : Array[1..8] of Byte;   // Information pertinien only to the sender of an encapsulation command
            Options : DInt;
         END_STRUCT;
         Data : Array[1..508] of Byte;
      END_STRUCT;
      receiveBuffer : Struct
         Header : Struct
            Command : Word;   // Encapsulation command
            Length : Int;   // Length, in bytes, of the command specific data portion of the message
            SessionHandle : DInt;   // Session identification
            Status : DInt;   // Status code
            Context : Array[1..8] of Byte;   // Information pertinien only to the sender of an encapsulation command
            Options : DInt;
         END_STRUCT;
         Data : Array[1..508] of Byte;
      END_STRUCT;
      currentResponse : Word;
      connectionStatus : Struct
         isDisconnected : Bool;
         isDisconnecting : Bool;
         isConnecting : Bool;
         isConnected : Bool;
         hasReceivedData : Bool;
         hasReceivedHeader : Bool;
      END_STRUCT;
      indexTag : Int := 0;
      currentCIPService : Byte;
      previousRequest : Bool;
      EnabledJ : Bool;
      ownInstance : DInt;
      ownSequence : DInt;
      randomGenerator : Struct   // [STRUCT] used to realize a pseudo random number
         m_w : DInt;
         m_z : DInt;
         Val : DInt;
         currentTime : Date_And_Time;
         currentMilliSeconds : Time;
      END_STRUCT;
   END_VAR
   VAR_TEMP
      indexTagName : Int;
      result : Int;
      itemLength : Int;   // contains the Length of the EIP packet
      overallLength : Int;   // contains the Length of the EIP packet
      tagNameLength : Int;   // contains the Length of the Tagname (in WORDS)
      unconnectedDataItemLength : Int;   // contains the Length of the unconnected data item
      baseIndexOuterCIPMessage : Int;   // contains the base index to the beginning of the outer CIP message
      baseIndexInnerCIPMessage : Int;   // contains the base index to the beginning of the inner CIP message
      receivedInstance : DInt;
      receivedSequence : DInt;
      receivedType : Word;
      valueIndex : Int;
      tagName : String[24];
      receivedValue : Byte;
      SrcAny : ANY;
      Source AT SrcAny : Struct
         ID : Byte;
         Typed : Byte;
         Amount : Int;
         Block : Int;
         Offset : Int;
      END_STRUCT;
   END_VAR
   VAR CONSTANT
      EIP_VENDOR_ID : Word := 1251;   // EtherNet/IP vendor ID 'Siemens AG'
      EIP_HEADER_LENGTH : Int := 24;   // EtherNet/IP Encapsulation Header length is 24 bytes
      EIP_PORT : Word := 44818;   // EtherNet/IP standard port is 44818 (0xAF12)
      RESULT_SUCCESS : Word := 16#0000;
      RESULT_IDLE : Word := 16#7000;
      RESULT_JOB_START : Word := 16#7001;
      RESULT_JOB_RUNNING : Word := 16#7002;
      RESULT_JOB_NOT_REQUIRED : Word := 16#80A3;
      RESULT_MORE_AVAIL : Word := 16#80B1;
      RESULT_REUSED_ID : Word := 16#8085;
      EIP_STATUS_OK : DInt := 16#0;   // EIP Status OK
      EIP_STATUS_TOOMANY_SESSIONS : DInt;   // EIP Status "more than 1 active session on the same TCP connection"
      EIP_STATUS_OUTOFRESSOURCES : DInt;   // EIP Status "does not have sufficient resources"
      EIP_STATUS_INVALID_SESSION_ID : DInt;   // EIP Status "Invalid Session ID"
      EIP_STATUS_PROTOCOL_ERROR : DInt;   // EIP Status "Protocol Version or Options mismatches"
      EIP_CMD_REG_SESSION : Word := 16#0065;   // EtherNet/IP Encapsulation Command "Register Session"
      EIP_CMD_UNREG_SESSION : Word := 16#0066;   // EtherNet/IP Encapsulation Command "Unregister Session"
      EIP_CMD_SEND_RR : Word := 16#006F;   // EtherNet/IP Encapsulation Command "Send RR Data"
      CIP_SRV_TABLEREAD : Byte := 16#4C;   // CIP Service Data Table Read
      CIP_SRV_TABLEWRITE : Byte := 16#4D;   // CIP Service Data Table Write
      CIP_SRV_TABLEREAD_FRAG : Byte := 16#52;   // CIP Service Fragmented Data Table Read
      CIP_SRV_TABLEWRITE_FRAG : Byte := 16#53;   // CIP Service Fragmented Data Table Write
      CIP_SRV_UNCONNECTED_SEND : Byte := 16#52;   // CIP Service Unconnected Send Data
      STATE_IDLE : Int := 1;
      STATE_INIT : Int := 2;
      STATE_CONNECTING : Int := 3;
      STATE_DISCONNECTING : Int := 4;
      STATE_SENDING : Int := 5;
      STATE_REGISTER_SESSION : Int := 6;
      STATE_UNREGISTER_SESSION : Int := 7;
      STATE_REGISTERING : Int := 8;
      STATE_UNREGISTERING : Int := 9;
      STATE_REGISTERED : Int := 10;
      STATE_SEND : Int := 11;
      STATE_RECEIVE_HEADER : Int := 12;
      STATE_RECEIVE_DATA : Int := 13;
      STATE_POWER_OFF : Int := 0;
      DT_BOOLEAN_ATOMIC : Int := 16#C1;
      DT_SINT_ATOMIC : Int := 16#C2;
      DT_INT_ATOMIC : Int := 16#C3;
      DT_DINT_ATOMIC : Int := 16#C4;
      DT_FLOAT_ATOMIC : Int := 16#CA;
      CIP_PATH_SEG_TYPE_CLASS : Byte := 16#20;
      CIP_PATH_SEG_TYPE_INSTANCE : Byte := 16#24;
      CIP_PATH_SEG_TYPE_ANSI : Byte := 16#91;
      CIP_PATH_SEG_TYPE_PORT : Byte := 16#01;
      CIP_ROUTE_SEG_LENGTH : Int := 4;
      CIP_ROUTE_PATH_LENGTH : Int := 1;
      CIP_TABLEREAD_LENGTH : Int := 6;
      CIP_UCSEND_HEADER_LENGTH : Int := 4;
      CIP_UCSEND_SEG_LENGTH : Int := 6;
      EIP_CMD_SEND_RR_SEG_LENGTH : Int := 16;
      CON_TYPE_TCP_V2 : Byte := 16#11;
      CON_TYPE_TCP_V4 : Byte := 11;
      CIP_GENSTS_SUCCESS : Byte := 16#00;
      CIP_GENSTS_PATH_SEG_ERROR : Byte := 16#04;
      CIP_GENSTS_PATH_DEST_UNKNOWN : Byte := 16#05;
      CIP_GENSTS_PARTIAL : Byte := 16#06;
      CIP_GENSTS_NOT_ENOUGH_DATA : Byte := 16#13;
      CIP_GENSTS_PATH_SIZE_MISMATCH : Byte := 16#26;
      CIP_GENSTS_DOESNT_EXIST : Byte := 16#16;
      CIP_GENSTS_GENERIC : Byte := 16#FF;
      CIP_SRVSTS_RANGE_EXCEED : Int := 16#2105;
   END_VAR
BEGIN
   //=============================================================================
   // Siemens AG
   // (c)Copyright 2016 All Rights Reserved
   //-----------------------------------------------------------------------------
   // Library: PutGet_Rockwell
   // Tested with: 319F-3PN/DP V2.8.6 and ControlLogix/Compactlogix V26
   // Engineering: TIA Portal V13 SP1 Upd 9
   // Restrictions: look into pdf
   // Requirements: 
   // Functionality: Get Put Values from to Rockwell CPU
   //-----------------------------------------------------------------------------
   // Change log table:
   // Version  Date            Expert in charge        Changes applied
   // 01.00.00 12.07.2016      Scheel                  initial version 
   // 01.00.01 20.10.2016      Scheel                  feat: add diagnostics and
   //                                                        indicators
   //                                                  style: remove duplicate
   //                                                         code segments
   //                                                  fix: connect will be
   //                                                       retriggered, when idle
   //                                                  refac: change of IP address
   //                                                         datatype to IP_V4
   //                                                  feat: add recognition of
   //                                                        CIP specific status
   //=============================================================================
   //

   //#########################################################################################
   // Pseudo Random number generator
   //
   //  This Random number function generator is based on multiplication and
   //  addition with overflow invented by George Marsaglia.
   //  The loss of information is intended.
   //  
   //  Wikipedia (https://en.wikipedia.org/wiki/Random_number_generation)
   //#########################################################################################
   //
   //Initialization of the variables using a time value as a seed
   //

   #randomGenerator.currentMilliSeconds := TIME_TCK();

   IF #randomGenerator.m_w = 0 OR #randomGenerator.m_z = 0 THEN
     #randomGenerator.m_w := T_CONV(TIME_TCK());    // using the milliseconds since the PLC has been powered on
     #randomGenerator.m_z := 13696;
   ELSE
     #randomGenerator.m_z := 36969 * DWORD_TO_DINT(DINT_TO_DWORD(#randomGenerator.m_z) AND 16#FFFF)
     + DWORD_TO_DINT(SHR(IN := DINT_TO_DWORD(#randomGenerator.m_z), N := 16));
     #randomGenerator.m_w := 18000 * DWORD_TO_DINT(DINT_TO_DWORD(#randomGenerator.m_w) AND 16#FFFF)
     + DWORD_TO_DINT(SHR(IN := DINT_TO_DWORD(#randomGenerator.m_w), N := 16));
     #randomGenerator.Val := DWORD_TO_DINT(SHL(IN := DINT_TO_DWORD(#randomGenerator.m_z), N := 16)) + #randomGenerator.m_w;  // 32-bit result */    
   END_IF;

   //assume sane state
   #Status := #RESULT_IDLE;
   #NewData := FALSE;

   #connect(ID := #connection.id,
            CONNECT := #connection);

   #disconnect(ID := #connection.id);


   IF NOT #Enable AND #EnabledJ THEN
     // Complete Restart detected 
     //
     #internalState := #STATE_UNREGISTER_SESSION;

   ELSIF #Enable AND NOT #EnabledJ THEN
     #internalState := #STATE_INIT;

   ELSE
     // Regular operation
     //
     CASE #internalState OF
       #STATE_POWER_OFF:
         //Preset the TCP connection information
         //
         IF #Config.connID = 0 THEN
           #Config.connID := DWORD_TO_WORD(DINT_TO_DWORD((#randomGenerator.Val MOD 2048) + 2048));
         END_IF;
         #connection.id := #Config.connID;

         #connection.connection_type := #CON_TYPE_TCP_V2;      //TCP connection
         #connection.local_device_id := #InterfaceId;
         #connection.active_est := TRUE;                //active connection (Client)

         #connection.local_tsap_id_len := 0;

         #connection.rem_staddr_len := 4;
         #connection.rem_staddr[1] := #IPv4[1];
         #connection.rem_staddr[2] := #IPv4[2];
         #connection.rem_staddr[3] := #IPv4[3];
         #connection.rem_staddr[4] := #IPv4[4];

         #connection.rem_tsap_id_len := 2;
         #connection.rem_tsap_id[1] := WORD_TO_BYTE(SHR(IN := #EIP_PORT, N := 8));
         #connection.rem_tsap_id[2] := WORD_TO_BYTE(#EIP_PORT AND W#16#FF);

         #ownInstance := 0;
         #ownSequence := 0;

         #internalState := #STATE_IDLE;

       #STATE_IDLE:

         // Action
         //
         #NewData := FALSE;

         // Transition 
         //IF NOT #connectionStatus.isConnected THEN
         //  #internalState := #STATE_INIT;
         IF #connectionStatus.isConnected AND #REQ AND NOT #previousRequest AND #Enable THEN
           #internalState := #STATE_SENDING;
           #Status := #RESULT_JOB_START;
         END_IF;


       #STATE_INIT:
         //Preset the TCP connection information
         //
         IF #Config.connID = 0 THEN
           #Config.connID := DWORD_TO_WORD(DINT_TO_DWORD((#randomGenerator.Val MOD 2048) + 2048));
         END_IF;
         #connection.id := #Config.connID;

         //Inserting Semaphore checking
         //
         //  Only issue a new connect, when there is no one is referencing the connection already
         //  Otherwise just skip that step and use the established connection
         //  

         IF #Config.references = 0 THEN
           #connection.connection_type := #CON_TYPE_TCP_V2;      //TCP connection
           #connection.local_device_id := #InterfaceId;
           #connection.active_est := TRUE;                //active connection (Client)

           #connection.local_tsap_id_len := 0;

           #connection.rem_staddr_len := 4;
           #connection.rem_staddr[1] := #IPv4[1];
           #connection.rem_staddr[2] := #IPv4[2];
           #connection.rem_staddr[3] := #IPv4[3];
           #connection.rem_staddr[4] := #IPv4[4];

           #connection.rem_tsap_id_len := 2;
           #connection.rem_tsap_id[1] := WORD_TO_BYTE(SHR(IN := #EIP_PORT, N := 8));
           #connection.rem_tsap_id[2] := WORD_TO_BYTE(          #EIP_PORT AND W#16#FF);


           //No connection established yet
           //  issue a new request
           #connect.REQ := TRUE;
           #internalState := #STATE_CONNECTING;
         ELSE
           #internalState := #STATE_IDLE;
           #connectionStatus.isConnected := TRUE;
         END_IF;
         #Config.references := #Config.references + 1;

         //Remember the currently active instance reference as my own instance identifier
         //  and reset the Sequence counter
         #ownInstance := #Config.references;
         #ownSequence := 0;

       #STATE_CONNECTING:

         IF #connect.STATUS = #RESULT_JOB_START THEN
           #connectionStatus.isConnecting := TRUE;

         ELSIF #connect.STATUS = #RESULT_IDLE THEN
           #connect.REQ := NOT #connect.REQ;

         ELSIF #connect.STATUS = #RESULT_JOB_RUNNING THEN
           #connect.REQ := FALSE;

         ELSIF #connect.STATUS = #RESULT_JOB_NOT_REQUIRED OR
           #connect.STATUS = #RESULT_SUCCESS
         THEN
           #connect.REQ := FALSE;
           #connectionStatus.isConnecting := FALSE;
           #connectionStatus.isConnected := TRUE;
           #connectionStatus.isDisconnected := FALSE;

           #internalState := #STATE_REGISTER_SESSION;

         ELSE
           // Throw error !
           //   Error in connect
           #Status := W#16#8100 OR (#connect.STATUS AND 16#00FF);   //Error in connecting
           #connect.REQ := FALSE;
           #internalState := #STATE_DISCONNECTING;
         END_IF;

       #STATE_REGISTER_SESSION:

         // SWAP (W#16#AFCD) = W#16#CDAF
         // 
         //  SHL(AFCD, 8) OR SHR(AFCD, 8)

         #sendBuffer.Header.Command :=(SHL(IN:=#EIP_CMD_REG_SESSION, N:= 8) OR SHR(IN:=#EIP_CMD_REG_SESSION, N:= 8)); //Command is RegisterSession (16#65)
         #sendBuffer.Header.Length := WORD_TO_INT(W#16#0400);          //Length of Data is 4 Bytes
         #sendBuffer.Header.SessionHandle := 0;
         #sendBuffer.Header.Status := 0;
         #sendBuffer.Header.Options := 0;
         //the Context will be a combination out of the own instance identifier
         //and a sequence number
         #sendBuffer.Header.Context[1] := DWORD_TO_BYTE(DINT_TO_DWORD(#ownInstance) AND DW#16#000000FF);
         #sendBuffer.Header.Context[2] := DWORD_TO_BYTE(SHR(IN := DINT_TO_DWORD(#ownInstance), N := 8) AND DW#16#000000FF);
         #sendBuffer.Header.Context[3] := DWORD_TO_BYTE(SHR(IN := DINT_TO_DWORD(#ownInstance), N := 16) AND DW#16#000000FF);
         #sendBuffer.Header.Context[4] := DWORD_TO_BYTE(SHR(IN := DINT_TO_DWORD(#ownInstance), N := 24) AND DW#16#000000FF);
         #sendBuffer.Header.Context[5] := DWORD_TO_BYTE(DINT_TO_DWORD(#ownSequence) AND DW#16#000000FF);
         #sendBuffer.Header.Context[6] := DWORD_TO_BYTE(SHR(IN := DINT_TO_DWORD(#ownSequence), N := 8) AND DW#16#000000FF);
         #sendBuffer.Header.Context[7] := DWORD_TO_BYTE(SHR(IN := DINT_TO_DWORD(#ownSequence), N := 16) AND DW#16#000000FF);
         #sendBuffer.Header.Context[8] := DWORD_TO_BYTE(SHR(IN := DINT_TO_DWORD(#ownSequence), N := 24) AND DW#16#000000FF);
         #sendBuffer.Data[1] := 16#01;                                 //Protocol Version V1.0

         //Checking the MuteEx
         IF #Config.instanceLock = 0 OR
           #Config.instanceLock = #ownInstance
         THEN
           //allowed to utilize, since instanceLock is either 0 or ownInstance
           #send(ID := #connection.id,
                 DATA := #sendBuffer);

           //Locking the MutEx
           #Config.instanceLock := #ownInstance;
           #send.LEN := #EIP_HEADER_LENGTH + 4;
           #send.REQ := TRUE;

           #internalState := #STATE_REGISTERING;
         ELSE
           ;
         END_IF;

       #STATE_REGISTERING:
         // Action
         // 

         //allowed to utilize, since instanceLock is either 0 or ownInstance
         #send(ID := #connection.id,
               DATA := #sendBuffer);

         // Transition
         // 
         IF #send.STATUS = #RESULT_JOB_START THEN
           ;
         ELSIF #send.STATUS = #RESULT_JOB_RUNNING THEN
           #send.REQ := FALSE;

         ELSIF #send.STATUS = #RESULT_IDLE THEN
           #send.REQ := NOT #send.REQ;

         ELSIF #send.STATUS = #RESULT_SUCCESS THEN
           #send.REQ := FALSE;
           #internalState := #STATE_RECEIVE_HEADER;
         ELSE
           // Throw error !
           //   in Registering
           #Status := W#16#8200 OR (#send.STATUS AND 16#00FF);   //Error in sending
           #send.REQ := FALSE;
           #internalState := #STATE_DISCONNECTING;
         END_IF;

       #STATE_SENDING:
         #sendBuffer.Header.Command := (SHL(IN:=#EIP_CMD_SEND_RR, N:=8) OR SHR(IN:=#EIP_CMD_SEND_RR, N:=8));       //Command is SendRRData (16#6F)
         //
         // overall Message length depends on the packet content and is therefore assigned later
         //
         // SWAP (DW#16#0102ABCD) = CDAB0201
         // 
         //   = SHL(<value>,24) OR (SHL(<value>, 8) AND DW#16#00FF0000) OR (SHR(<value>, 8) AND DW#16#0000FF00) OR SHR(<value>,24)

         //#sendBuffer.Header.SessionHandle := DWORD_TO_DINT(SWAP(DINT_TO_DWORD(#Config.currentSessionID)));
         #sendBuffer.Header.SessionHandle := DWORD_TO_DINT(SHL(IN := DINT_TO_DWORD(#Config.currentSessionID), N := 24) OR
                                                           (SHL(IN := DINT_TO_DWORD(#Config.currentSessionID), N := 8) AND DW#16#00FF0000) OR
                                                           (SHR(IN := DINT_TO_DWORD(#Config.currentSessionID), N := 8) AND DW#16#0000FF00) OR
                                                           SHR(IN := DINT_TO_DWORD(#Config.currentSessionID), N := 24));

         ;
         #sendBuffer.Header.Status := 0;
         #sendBuffer.Header.Options := 0;
         //the Context will be a combination out of the own instance identifier
         //and a sequence number
         #sendBuffer.Header.Context[1] := DWORD_TO_BYTE(DINT_TO_DWORD(#ownInstance) AND DW#16#000000FF);
         #sendBuffer.Header.Context[2] := DWORD_TO_BYTE(SHR(IN := DINT_TO_DWORD(#ownInstance), N := 8) AND DW#16#000000FF);
         #sendBuffer.Header.Context[3] := DWORD_TO_BYTE(SHR(IN := DINT_TO_DWORD(#ownInstance), N := 16) AND DW#16#000000FF);
         #sendBuffer.Header.Context[4] := DWORD_TO_BYTE(SHR(IN := DINT_TO_DWORD(#ownInstance), N := 24) AND DW#16#000000FF);
         #sendBuffer.Header.Context[5] := DWORD_TO_BYTE(DINT_TO_DWORD(#ownSequence) AND DW#16#000000FF);
         #sendBuffer.Header.Context[6] := DWORD_TO_BYTE(SHR(IN := DINT_TO_DWORD(#ownSequence), N := 8) AND DW#16#000000FF);
         #sendBuffer.Header.Context[7] := DWORD_TO_BYTE(SHR(IN := DINT_TO_DWORD(#ownSequence), N := 16) AND DW#16#000000FF);
         #sendBuffer.Header.Context[8] := DWORD_TO_BYTE(SHR(IN := DINT_TO_DWORD(#ownSequence), N := 24) AND DW#16#000000FF);
         //CIP specific data
         #sendBuffer.Data[1] := 16#0;                                 //CIP Interface handle
         #sendBuffer.Data[2] := 16#0;
         #sendBuffer.Data[3] := 16#0;
         #sendBuffer.Data[4] := 16#0;

         #sendBuffer.Data[5] := 16#0;                                  //Timeout
         #sendBuffer.Data[6] := 16#0;

         #sendBuffer.Data[7] := 16#2;                                  //Items
         #sendBuffer.Data[8] := 16#0;

         #sendBuffer.Data[9] := 16#0;                                  //Null address item
         #sendBuffer.Data[10] := 16#0;
         #sendBuffer.Data[11] := 16#0;                                  //Null address item Length = 0
         #sendBuffer.Data[12] := 16#0;

         #sendBuffer.Data[13] := 16#B2;                                  //Unconnected data item
         #sendBuffer.Data[14] := 16#0;
         //Item Length needs to be added, but since that depends on the content,
         //it will will be assigned later. It occupies 2 Bytes, thus the outer CIP Message 
         //starts at offset 17 into the Data (1 based counting)
         //
         #baseIndexOuterCIPMessage := 17;

         //CIP Message
         //  here a decision needs to be made
         //  In case Slot is -1 a direct connection is assumed, such as for a CompactLogix, this means no
         //  further route segments are necessary
         //  In case Slot is anywhere between 0 and 16 a route segment is required, since the CPU is not
         //  identical to the ethernet interface, as in a ControlLogix L5, L6, L7 series system

         //Length of the following Path segment depends only on the length of the Tagname measured in WORDS
         // plus 1 WORD for the segment encoding information
         //
         #tagName := #Tag."Name";
         #tagNameLength := ((LEN(#tagName) + 1) / 2) * 2;

         //
         //  Prelude
         //
         //In case the slot information is negative (-1) there is no additional path segment
         //Any other slot value requires routing information, which need to be added
         //  this means the preparation of offsets and header needs to be done, before
         //  the common part of copying the value to the packet can take place
         IF #Slot = -1 THEN
           //directly connected (onboard) Ethernet interface
           //
           #baseIndexInnerCIPMessage := #baseIndexOuterCIPMessage;

         ELSE
           //not directly connected (through external) Ethernet interface
           //
           //  preparing offsets for length calculation as well as header
           //  There is a 10 byte segment before the tag value segment
           #baseIndexInnerCIPMessage := #baseIndexOuterCIPMessage + 10;

           #sendBuffer.Data[#baseIndexOuterCIPMessage] := #CIP_SRV_UNCONNECTED_SEND;  //CIP service = UNCONNECTED_SEND_DATA = 16#52
           #sendBuffer.Data[#baseIndexOuterCIPMessage + 1] := 2;                                     //Path Size is constant 2 WORDS

           #sendBuffer.Data[#baseIndexOuterCIPMessage + 2] := #CIP_PATH_SEG_TYPE_CLASS;              //Path Type = Class Segment
           #sendBuffer.Data[#baseIndexOuterCIPMessage + 3] := 16#06;                                 //Class = ConnectionManager (16#06)

           #sendBuffer.Data[#baseIndexOuterCIPMessage + 4] := #CIP_PATH_SEG_TYPE_INSTANCE;           //Path Type = Instance Segment
           #sendBuffer.Data[#baseIndexOuterCIPMessage + 5] := 16#01;                                 //Instance =Instance 1 (16#01)

           //Encapsulated CIP Message
           //
           #sendBuffer.Data[#baseIndexOuterCIPMessage + 6] := 16#07;                                 //Priority combined with TimeTick (= 16#07)
           #sendBuffer.Data[#baseIndexOuterCIPMessage + 7] := INT_TO_BYTE(233);                     //???

         END_IF;

         //
         // tag value segment
         // 

         #sendBuffer.Data[#baseIndexInnerCIPMessage] := #CIP_SRV_TABLEREAD;                        //CIP service = DATA_TABLE_READ = 16#4C

         #sendBuffer.Data[#baseIndexInnerCIPMessage + 1] := DINT_TO_BYTE(#tagNameLength / 2 + 1);  //Path Size
         #sendBuffer.Data[#baseIndexInnerCIPMessage + 2] := #CIP_PATH_SEG_TYPE_ANSI;               //Path Type = ANSI Extended Symbol Segment

         //Copy In
         #tagName := #Tag."Name";
         #sendBuffer.Data[#baseIndexInnerCIPMessage + 3] := INT_TO_BYTE(LEN(#tagName));   //TagName Length (bytes)
         FOR #indexTagName := 1 TO BYTE_TO_INT(#sendBuffer.Data[#baseIndexInnerCIPMessage + 3]) DO
           #sendBuffer.Data[#baseIndexInnerCIPMessage + 3 + #indexTagName] := CHAR_TO_BYTE(S_CONV(MID(IN := #tagName, L := 1, P := #indexTagName)));
         END_FOR;

         //in case the tag name has an odd (uneven) length the path segment content needs to be padded to be WORD aligned
         //
         #indexTagName := #indexTagName - 1;
         IF #indexTagName MOD 2 <> 0 THEN
           #indexTagName := #indexTagName + 1;
           #sendBuffer.Data[#baseIndexInnerCIPMessage + 3 + #indexTagName] := 0;
         END_IF;

         //Command Specific information
         //

         #sendBuffer.Data[#baseIndexInnerCIPMessage + 4 + #indexTagName] := INT_TO_BYTE(#Tag.Count);//1;                  //Number of Items
         #sendBuffer.Data[#baseIndexInnerCIPMessage + 5 + #indexTagName] := WORD_TO_BYTE(SHR(IN := INT_TO_WORD(#Tag.Count), N := 8) AND W#16#00FF);//0;

         #itemLength := #tagNameLength + #CIP_TABLEREAD_LENGTH;

         //
         // Closure
         //

         IF #Slot = -1 THEN
           #unconnectedDataItemLength := #itemLength;
         ELSE
           #sendBuffer.Data[#baseIndexOuterCIPMessage + 8] := WORD_TO_BYTE(DINT_TO_WORD(#itemLength));                  //Unconnected data item Length
           #sendBuffer.Data[#baseIndexOuterCIPMessage + 9] := WORD_TO_BYTE(SHL(IN := DINT_TO_WORD(#itemLength), N := 8));  //Unconnected data item Length

           //Routing Information
           #sendBuffer.Data[#baseIndexInnerCIPMessage + #itemLength    ] := INT_TO_BYTE(#CIP_ROUTE_PATH_LENGTH);
           #sendBuffer.Data[#baseIndexInnerCIPMessage + #itemLength + 1] := 0;

           #sendBuffer.Data[#baseIndexInnerCIPMessage + #itemLength + 2] := #CIP_PATH_SEG_TYPE_PORT;
           #sendBuffer.Data[#baseIndexInnerCIPMessage + #itemLength + 3] := INT_TO_BYTE(#Slot);

           #unconnectedDataItemLength :=   #itemLength
                                         + #CIP_ROUTE_SEG_LENGTH
                                         + #CIP_UCSEND_HEADER_LENGTH
                                         + #CIP_UCSEND_SEG_LENGTH;
         END_IF;

         //Length of the unconnected data item depends on the content of the package
         //
         #sendBuffer.Data[15] := WORD_TO_BYTE(DINT_TO_WORD(#unconnectedDataItemLength));                //Unconnected data item Length
         #sendBuffer.Data[16] := WORD_TO_BYTE(SHL(IN := DINT_TO_WORD(#unconnectedDataItemLength), N := 8));  //Unconnected data item Length


         #sendBuffer.Header.Length := WORD_TO_INT(SHL(IN := INT_TO_WORD(#unconnectedDataItemLength + #EIP_CMD_SEND_RR_SEG_LENGTH), N:=8) OR
                                                  SHR(IN := INT_TO_WORD(#unconnectedDataItemLength + #EIP_CMD_SEND_RR_SEG_LENGTH), N:=8));    //Length of Data


         //Checking the MuteEx
         IF #Config.instanceLock = 0 OR
           #Config.instanceLock = #ownInstance
         THEN
           //Locking the MutEx
           #Config.instanceLock := #ownInstance;
           #send.LEN := DINT_TO_INT(#EIP_HEADER_LENGTH + #unconnectedDataItemLength + #EIP_CMD_SEND_RR_SEG_LENGTH);
           #send.REQ := TRUE;

           //allowed to utilize, since instanceLock is either 0 or ownInstance
           #send(ID := #connection.id,
                 DATA := #sendBuffer);

           #internalState := #STATE_SEND;
         ELSE
           ;
         END_IF;
         #Status := #RESULT_JOB_RUNNING;

       #STATE_SEND:
         // Action
         // 
         // assume job is still running
         #Status := #RESULT_JOB_RUNNING;

         #send(ID := #connection.id,
               DATA := #sendBuffer);

         // Transition
         //
         IF #send.STATUS = #RESULT_JOB_START THEN
           ;
         ELSIF #send.STATUS = #RESULT_IDLE THEN
           #send.REQ := NOT #send.REQ;

         ELSIF #send.STATUS = #RESULT_JOB_RUNNING THEN
           #send.REQ := FALSE;

         ELSIF #send.STATUS = #RESULT_SUCCESS THEN
           #send.REQ := FALSE;
           #internalState := #STATE_RECEIVE_HEADER;
         ELSE
           // Throw error !
           // 
           #Status := W#16#8200 OR (#send.STATUS AND 16#00FF);
           #send.REQ := FALSE;
           #internalState := #STATE_DISCONNECTING;
         END_IF;


       #STATE_RECEIVE_HEADER:
         // Action
         // Receive Header data
         // 
         #receive(EN_R := (#ownInstance = #Config.instanceLock),
                  ID := #connection.id,
                  LEN := #EIP_HEADER_LENGTH,
                  DATA := #receiveBuffer.Header);


         // Transition
         // Header received --> STATE_RECEIVE_DATA
         // Invalid Data --> IDLE
         // Error --> INIT
         IF #receive.NDR OR #receive.STATUS = #RESULT_SUCCESS THEN
           IF #receiveBuffer.Header.Length = 0 THEN
             //Unlocking MuteEx
             #Config.instanceLock := 0;
             #internalState := #STATE_IDLE;
           ELSE
             #internalState := #STATE_RECEIVE_DATA;
           END_IF;

         ELSIF #receive.STATUS <> #RESULT_IDLE AND
           #receive.STATUS <> #RESULT_JOB_RUNNING AND
           #receive.STATUS <> #RESULT_JOB_START AND
           #receive.STATUS <> #RESULT_SUCCESS
         THEN
           #Status := W#16#8300 OR (#receive.STATUS AND 16#00FF);
           #internalState := #STATE_IDLE;
         ELSE
           ;
         END_IF;

       #STATE_RECEIVE_DATA:
         // Action
         // Receive Data
         // 
         // assume job is still running
         #Status := #RESULT_JOB_RUNNING;

         #receive(EN_R := (#ownInstance = #Config.instanceLock),
                  ID := #connection.id,
                  LEN := WORD_TO_INT((SHL(IN:=INT_TO_WORD(#receiveBuffer.Header.Length),N:= 8) OR
                                      SHR(IN:=INT_TO_WORD(#receiveBuffer.Header.Length),N:= 8))),
                  DATA := #receiveBuffer.Data);

         // Transition
         // Header received --> STATE_RECEIVE_DATA
         // Invalid Data --> IDLE
         // Error --> INIT

         IF #receive.NDR OR #receive.STATUS = #RESULT_SUCCESS THEN
           // Decode Response
           // 
           #currentResponse := (SHL(IN:=#receiveBuffer.Header.Command, N:=8) OR
                                SHR(IN:=#receiveBuffer.Header.Command, N:=8));

           //the Context will be a combination out of the own instance identifier
           //and a sequence number
           #receivedInstance := DWORD_TO_DINT(SHL(IN := BYTE_TO_DWORD(#receiveBuffer.Header.Context[4]), N := 24) OR
                                              SHL(IN := BYTE_TO_DWORD(#receiveBuffer.Header.Context[3]), N := 16) OR
                                              SHL(IN := BYTE_TO_DWORD(#receiveBuffer.Header.Context[2]), N := 8) OR
                                              BYTE_TO_DWORD(#receiveBuffer.Header.Context[1]));

           #receivedSequence := DWORD_TO_DINT(SHL(IN := BYTE_TO_DWORD(#receiveBuffer.Header.Context[8]), N := 24) OR
                                              SHL(IN := BYTE_TO_DWORD(#receiveBuffer.Header.Context[7]), N := 16) OR
                                              SHL(IN := BYTE_TO_DWORD(#receiveBuffer.Header.Context[6]), N := 8) OR
                                              BYTE_TO_DWORD(#receiveBuffer.Header.Context[5]));

           IF #currentResponse = #EIP_CMD_REG_SESSION THEN
             //Response to RegisterSession received
             // retrieve the SessionID (SessionHandle)
             IF #receiveBuffer.Header.Status = #EIP_STATUS_OK THEN
               // SWAP (DW#16#0102ABCD) = CDAB0201
               // 
               //   = SHL(<value>,24) OR (SHL(<value>, 8) AND DW#16#00FF0000) OR (SHR(<value>, 8) AND DW#16#0000FF00) OR SHR(<value>,24)

               //#Config.currentSessionID := DWORD_TO_DINT(SWAP(DINT_TO_DWORD(#receiveBuffer.Header.SessionHandle)));
               #Config.currentSessionID := DWORD_TO_DINT( SHL(IN:=DINT_TO_DWORD(#receiveBuffer.Header.SessionHandle),N:=24) OR
                                                         (SHL(IN:=DINT_TO_DWORD(#receiveBuffer.Header.SessionHandle),N:= 8) AND DW#16#00FF0000) OR
                                                         (SHR(IN:=DINT_TO_DWORD(#receiveBuffer.Header.SessionHandle),N:= 8) AND DW#16#0000FF00) OR
                                                          SHR(IN:=DINT_TO_DWORD(#receiveBuffer.Header.SessionHandle),N:=24));
                #Status := #RESULT_SUCCESS;
              ELSE
                // inform the user about it
                // 
                #Status := W#16#7100 OR DWORD_TO_WORD((SHR(IN := DINT_TO_DWORD(#receiveBuffer.Header.Status), N := 24)));

                //Cleaning up internal information and
                //gracefully disconnect
                IF #Config.currentSessionID = 0 THEN
                  // a previous session hasn't been established --> only disconnecting
                  #internalState := #STATE_DISCONNECTING;
                ELSE
                  // previous session existed (somehow) --> unregister before disconnecting
                  #internalState := #STATE_UNREGISTER_SESSION;
                END_IF;
              END_IF;

           ELSIF #currentResponse = #EIP_CMD_SEND_RR THEN
             //Response to Send RR Data received
             // determine Status of transmission
             // retrieve TagValue and DataType
             IF #receiveBuffer.Header.Status = #EIP_STATUS_OK THEN
               #itemLength := WORD_TO_INT(SHL(IN := BYTE_TO_WORD(#receiveBuffer.Data[16]), N := 8) OR BYTE_TO_WORD(#receiveBuffer.Data[15]));
               #currentCIPService := (#receiveBuffer.Data[17]);
               IF #currentCIPService = (#CIP_SRV_TABLEREAD OR 16#80) AND
                 #receivedInstance = #ownInstance AND
                 #receivedSequence = #ownSequence
               THEN
                 //Check the status of the variable request
                 //  it may have failed on us (<>0)
                 //  
                 IF #receiveBuffer.Data[19] = #CIP_GENSTS_SUCCESS THEN

                   #receivedType := SHL(IN := BYTE_TO_WORD(#receiveBuffer.Data[22]), N := 8) OR
                                              BYTE_TO_WORD(#receiveBuffer.Data[21]);

                   #SrcAny := #receiveBuffer.Data[23];
                   #Source.Amount := #Tag.Count;

                   CASE WORD_TO_INT(#receivedType) OF
                     #DT_BOOLEAN_ATOMIC:
                       #Source.Typed := B#16#02;           // S7 type is BYTE

                       #result := BLKMOV(SRCBLK := #SrcAny,
                                         DSTBLK => #Value);
                     #DT_SINT_ATOMIC:

                       #Source.Typed := B#16#02;           // S7 type is BYTE

                       #result := BLKMOV(SRCBLK := #SrcAny,
                                         DSTBLK => #Value);
                     #DT_INT_ATOMIC:
                       #valueIndex := 0;
                       WHILE #valueIndex <= (#itemLength - 6) DO

                         // swap the received value
                         #receivedValue := #receiveBuffer.Data[24 + #valueIndex];
                         #receiveBuffer.Data[24 + #valueIndex] := #receiveBuffer.Data[23 + #valueIndex];
                         #receiveBuffer.Data[23 + #valueIndex] := #receivedValue;

                         #valueIndex := #valueIndex + 2;
                       END_WHILE;

                       #Source.Typed := B#16#05;

                       #result := BLKMOV(SRCBLK := #SrcAny,
                                         DSTBLK => #Value);
                     #DT_DINT_ATOMIC:
                       #valueIndex := 0;
                       WHILE #valueIndex <= (#itemLength - 6) DO

                         // swap the received value
                         #receivedValue := #receiveBuffer.Data[26 + #valueIndex];
                         #receiveBuffer.Data[26 + #valueIndex] := #receiveBuffer.Data[23 + #valueIndex];
                         #receiveBuffer.Data[23 + #valueIndex] := #receivedValue;

                         #receivedValue := #receiveBuffer.Data[25 + #valueIndex];
                         #receiveBuffer.Data[25 + #valueIndex] := #receiveBuffer.Data[24 + #valueIndex];
                         #receiveBuffer.Data[24 + #valueIndex] := #receivedValue;

                         #valueIndex := #valueIndex + 4;
                       END_WHILE;

                       #Source.Typed := B#16#07;

                       #result := BLKMOV(SRCBLK := #SrcAny,
                                         DSTBLK => #Value);

                     #DT_FLOAT_ATOMIC:
                       #valueIndex := 0;
                       WHILE #valueIndex <= (#itemLength - 6) DO

                         // swap the received value
                         #receivedValue := #receiveBuffer.Data[26 + #valueIndex];
                         #receiveBuffer.Data[26 + #valueIndex] := #receiveBuffer.Data[23 + #valueIndex];
                         #receiveBuffer.Data[23 + #valueIndex] := #receivedValue;

                         #receivedValue := #receiveBuffer.Data[25 + #valueIndex];
                         #receiveBuffer.Data[25 + #valueIndex] := #receiveBuffer.Data[24 + #valueIndex];
                         #receiveBuffer.Data[24 + #valueIndex] := #receivedValue;

                         #valueIndex := #valueIndex + 4;
                       END_WHILE;

                       #Source.Typed := B#16#08;

                       #result := BLKMOV(SRCBLK := #SrcAny,
                                         DSTBLK => #Value);
                     ELSE
                       // throw warning
                       #Status := 16#71A3; //Unknown data type
                     END_CASE;

                   // show successful result
                   //
                   #Status := #RESULT_SUCCESS;

                   #NewData := TRUE;
                   IF #ownSequence = -1 THEN
                     #ownSequence := #ownSequence + 2;
                   ELSE
                     #ownSequence := #ownSequence + 1;
                   END_IF;
                 ELSIF #receiveBuffer.Data[19] = #CIP_GENSTS_PATH_DEST_UNKNOWN OR
                   #receiveBuffer.Data[19] = #CIP_GENSTS_PATH_SEG_ERROR
                 THEN
                   // throw warning
                   #Status := W#16#7200 OR #receiveBuffer.Data[19];

                 ELSIF #receiveBuffer.Data[19] = #CIP_GENSTS_GENERIC THEN
                   #Status := W#16#7300 OR #receiveBuffer.Data[22];
                 ELSE
                   // throw warning
                   #Status := W#16#72FF;  //Unknown error code
                 END_IF;

                 ELSIF #currentCIPService = (#CIP_SRV_TABLEREAD_FRAG OR 16#80) THEN
                   #Status := W#16#7300 OR #receiveBuffer.Data[19];

                 ELSE
                   // throw warning
                   //   unexpected answer from host - ignoring it
                   #Status := W#16#8A00 OR #currentCIPService;
                 END_IF;
             ELSE
               // inform the user about it
               // 
               #Status := W#16#7100 OR DWORD_TO_WORD((SHR(IN := DINT_TO_DWORD(#receiveBuffer.Header.Status), N := 24)));

               //Cleaning up internal information and
               //gracefully disconnect
               IF #Config.currentSessionID = 0 THEN
                 // a previous session hasn't been established --> only disconnecting
                 #internalState := #STATE_DISCONNECTING;
               ELSE
                 // previous session existed (somehow) --> unregister before disconnecting
                 #internalState := #STATE_UNREGISTER_SESSION;
               END_IF;
             END_IF;
           ELSE
             //Unknown/ Unhandled Response received
             //  ignoring it
             #Status := W#16#8B00 OR #currentResponse;

             //#Config.currentSessionID := 0;
             //#internalState := #STATE_DISCONNECTING;
           END_IF;

           #receiveBuffer.Header.Length := 0;

           //Unlocking MuteEx
           #Config.instanceLock := 0;

           #internalState := #STATE_IDLE;
         ELSIF #receive.STATUS <> #RESULT_IDLE AND
           #receive.STATUS <> #RESULT_JOB_RUNNING AND
           #receive.STATUS <> #RESULT_JOB_START AND
           #receive.STATUS <> #RESULT_SUCCESS
         THEN
           #Status := W#16#8300 OR (#receive.STATUS AND 16#00FF);
           #internalState := #STATE_IDLE;
         ELSE
           //Nothing to do, just wait here
           ;
         END_IF;

       #STATE_UNREGISTER_SESSION:
         IF #Config.references = 1 THEN

           #sendBuffer.Header.Command := SHL(IN:=#EIP_CMD_UNREG_SESSION, N:= 8) OR
                                         SHR(IN:=#EIP_CMD_UNREG_SESSION, N:= 8);   //Command is RegisterSession (16#66)
           #sendBuffer.Header.Length := WORD_TO_INT(SHL(IN := INT_TO_WORD(#send.LEN - #EIP_HEADER_LENGTH),N:=8) OR
                                                    SHR(IN := INT_TO_WORD(#send.LEN - #EIP_HEADER_LENGTH),N:=8));    //Length of Data is 4 Bytes

           // SWAP (DW#16#0102ABCD) = CDAB0201
           // 
           //   = SHL(<value>,24) OR (SHL(<value>, 8) AND DW#16#00FF0000) OR (SHR(<value>, 8) AND DW#16#0000FF00) OR SHR(<value>,24)

